LIN {X 0,Y 354.811,Z 376.286,A -85,B 0,C 180,E1 -13642.402,E2 -13642.402} C_VEL
LIN {X 0,Y 354.817,Z 376.286,A -85,B 0,C 180,E1 -13644.524,E2 -13644.524} C_VEL
LIN {X 0,Y 354.143,Z 376.373,A -85,B 0,C 180,E1 -13645.473,E2 -13645.473} C_VEL
LIN {X 0,Y 351.322,Z 376.725,A -85,B 0,C 180,E1 -13647.018,E2 -13647.018} C_VEL
LIN {X 0,Y 348.61,Z 377.585,A -85,B 0,C 180,E1 -13648.572,E2 -13648.572} C_VEL
LIN {X 0,Y 348.11,Z 378.744,A -85,B 0,C 180,E1 -13649.518,E2 -13649.518} C_VEL
LIN {X 0,Y 347.833,Z 384.152,A -85,B 0,C 180,E1 -13652.752,E2 -13652.752} C_VEL
LIN {X 0,Y 347.434,Z 390.956,A -85,B 0,C 180,E1 -13656.768,E2 -13656.768} C_VEL
LIN {X 0,Y 347.187,Z 397.381,A -85,B 0,C 180,E1 -13660.488,E2 -13660.488} C_VEL
LIN {X 0,Y 346.96,Z 403.814,A -85,B 0,C 180,E1 -13664.13,E2 -13664.13} C_VEL
LIN {X 0,Y 346.774,Z 410.819,A -85,B 0,C 180,E1 -13668.01,E2 -13668.01} C_VEL
LIN {X 0,Y 346.782,Z 411.483,A -85,B 0,C 180,E1 -13668.27,E2 -13668.27} C_VEL
LIN {X 0,Y 348.09,Z 422.89,A -85,B 0,C 180,E1 -13669.015,E2 -13669.015} C_VEL
LIN {X 0,Y 348.747,Z 429.335,A -85,B 0,C 180,E1 -13669.55,E2 -13669.55} C_VEL
LIN {X 0,Y 348.245,Z 439.424,A -85,B 0,C 180,E1 -13670.562,E2 -13670.562} C_VEL
LIN {X 0,Y 347.847,Z 448.426,A -85,B 0,C 180,E1 -13671.723,E2 -13671.723} C_VEL
LIN {X 0,Y 347.615,Z 456.417,A -85,B 0,C 180,E1 -13673.032,E2 -13673.032} C_VEL
LIN {X 0,Y 347.324,Z 463.366,A -85,B 0,C 180,E1 -13674.484,E2 -13674.484} C_VEL
LIN {X 0,Y 347.115,Z 468.718,A -85,B 0,C 180,E1 -13675.936,E2 -13675.936} C_VEL
LIN {X 0,Y 346.768,Z 473.44,A -85,B 0,C 180,E1 -13677.677,E2 -13677.677} C_VEL
LIN {X 0,Y 346.735,Z 475.64,A -85,B 0,C 180,E1 -13678.839,E2 -13678.839} C_VEL
LIN {X 0,Y 346.756,Z 477.156,A -85,B 0,C 180,E1 -13680,E2 -13680} C_VEL
LIN {X 0,Y 346.825,Z 478.018,A -85,B 0,C 180,E1 -13681.161,E2 -13681.161} C_VEL
LIN {X 0,Y 346.995,Z 478.228,A -85,B 0,C 180,E1 -13682.322,E2 -13682.322} C_VEL
LIN {X 0,Y 347.302,Z 477.789,A -85,B 0,C 180,E1 -13683.48,E2 -13683.48} C_VEL
LIN {X 0,Y 347.777,Z 476.691,A -85,B 0,C 180,E1 -13684.636,E2 -13684.636} C_VEL
LIN {X 0,Y 348.649,Z 473.789,A -85,B 0,C 180,E1 -13686.365,E2 -13686.365} C_VEL
LIN {X 0,Y 349.587,Z 469.338,A -85,B 0,C 180,E1 -13688.09,E2 -13688.09} C_VEL
LIN {X 0,Y 350.585,Z 464.252,A -85,B 0,C 180,E1 -13689.52,E2 -13689.52} C_VEL
LIN {X 0,Y 351.785,Z 457.649,A -85,B 0,C 180,E1 -13690.941,E2 -13690.941} C_VEL
LIN {X 0,Y 353.113,Z 449.6,A -85,B 0,C 180,E1 -13692.289,E2 -13692.289} C_VEL
LIN {X 0,Y 354.289,Z 439.873,A -85,B 0,C 180,E1 -13693.587,E2 -13693.587} C_VEL
LIN {X 0,Y 352.987,Z 431.307,A -85,B 0,C 180,E1 -13694.705,E2 -13694.705} C_VEL
LIN {X 0,Y 349.84,Z 420.355,A -85,B 0,C 180,E1 -13696.038,E2 -13696.038} C_VEL
LIN {X 0,Y 348.708,Z 416.833,A -85,B 0,C 180,E1 -13696.465,E2 -13696.465} C_VEL
LIN {X 0,Y 349.163,Z 413.41,A -85,B 0,C 180,E1 -13698.91,E2 -13698.91} C_VEL
LIN {X 0,Y 349.782,Z 408.791,A -85,B 0,C 180,E1 -13702.443,E2 -13702.443} C_VEL
LIN {X 0,Y 350.665,Z 404.335,A -85,B 0,C 180,E1 -13706.163,E2 -13706.163} C_VEL
LIN {X 0,Y 351.349,Z 401.637,A -85,B 0,C 180,E1 -13708.69,E2 -13708.69} C_VEL
LIN {X 0,Y 351.882,Z 399.265,A -85,B 0,C 180,E1 -13711.285,E2 -13711.285} C_VEL
LIN {X 0,Y 352.025,Z 397.313,A -85,B 0,C 180,E1 -13713.987,E2 -13713.987} C_VEL
LIN {X 0,Y 352.035,Z 395.851,A -85,B 0,C 180,E1 -13717.007,E2 -13717.007} C_VEL
LIN {X 0,Y 352.049,Z 395.224,A -85,B 0,C 180,E1 -13719.704,E2 -13719.704} C_VEL
LIN {X 0,Y 352.23,Z 395.281,A -85,B 0,C 180,E1 -13722.719,E2 -13722.719} C_VEL
LIN {X 0,Y 352.561,Z 396.33,A -85,B 0,C 180,E1 -13725.859,E2 -13725.859} C_VEL
LIN {X 0,Y 353.162,Z 398.551,A -85,B 0,C 180,E1 -13729.131,E2 -13729.131} C_VEL
LIN {X 0,Y 353.976,Z 402.286,A -85,B 0,C 180,E1 -13732.578,E2 -13732.578} C_VEL
LIN {X 0,Y 355.113,Z 406.755,A -85,B 0,C 180,E1 -13735.665,E2 -13735.665} C_VEL
LIN {X 0,Y 355.806,Z 411.281,A -85,B 0,C 180,E1 -13738.141,E2 -13738.141} C_VEL
LIN {X 0,Y 355.791,Z 413.274,A -85,B 0,C 180,E1 -13739.097,E2 -13739.097} C_VEL
LIN {X 0,Y 354.038,Z 419.488,A -85,B 0,C 180,E1 -13741.548,E2 -13741.548} C_VEL
LIN {X 0,Y 351.605,Z 429.59,A -85,B 0,C 180,E1 -13745.181,E2 -13745.181} C_VEL
LIN {X 0,Y 350.041,Z 439.051,A -85,B 0,C 180,E1 -13748.273,E2 -13748.273} C_VEL
LIN {X 0,Y 352.668,Z 451.93,A -85,B 0,C 180,E1 -13749.147,E2 -13749.147} C_VEL
LIN {X 0,Y 353.713,Z 462.761,A -85,B 0,C 180,E1 -13749.95,E2 -13749.95} C_VEL
LIN {X 0,Y 353.653,Z 473.701,A -85,B 0,C 180,E1 -13750.859,E2 -13750.859} C_VEL
LIN {X 0,Y 352.881,Z 482.708,A -85,B 0,C 180,E1 -13751.719,E2 -13751.719} C_VEL
LIN {X 0,Y 351.276,Z 493.812,A -85,B 0,C 180,E1 -13752.986,E2 -13752.986} C_VEL
LIN {X 0,Y 350.022,Z 502.896,A -85,B 0,C 180,E1 -13754.272,E2 -13754.272} C_VEL
LIN {X 0,Y 348.637,Z 512.75,A -85,B 0,C 180,E1 -13756.001,E2 -13756.001} C_VEL
LIN {X 0,Y 347.733,Z 520.726,A -85,B 0,C 180,E1 -13757.748,E2 -13757.748} C_VEL
LIN {X 0,Y 346.937,Z 527.128,A -85,B 0,C 180,E1 -13759.495,E2 -13759.495} C_VEL
LIN {X 0,Y 346.618,Z 532.253,A -85,B 0,C 180,E1 -13761.253,E2 -13761.253} C_VEL
LIN {X 0,Y 346.518,Z 536.239,A -85,B 0,C 180,E1 -13763.01,E2 -13763.01} C_VEL
LIN {X 0,Y 346.434,Z 538.314,A -85,B 0,C 180,E1 -13764.178,E2 -13764.178} C_VEL
LIN {X 0,Y 346.456,Z 539.912,A -85,B 0,C 180,E1 -13765.346,E2 -13765.346} C_VEL
LIN {X 0,Y 346.562,Z 541.078,A -85,B 0,C 180,E1 -13766.512,E2 -13766.512} C_VEL
LIN {X 0,Y 346.686,Z 541.834,A -85,B 0,C 180,E1 -13767.676,E2 -13767.676} C_VEL
LIN {X 0,Y 346.736,Z 542.119,A -85,B 0,C 180,E1 -13768.838,E2 -13768.838} C_VEL
LIN {X 0,Y 346.701,Z 541.952,A -85,B 0,C 180,E1 -13770,E2 -13770} C_VEL
LIN {X 0,Y 346.742,Z 541.378,A -85,B 0,C 180,E1 -13771.161,E2 -13771.161} C_VEL
LIN {X 0,Y 346.843,Z 540.334,A -85,B 0,C 180,E1 -13772.322,E2 -13772.322} C_VEL
LIN {X 0,Y 346.663,Z 537.849,A -85,B 0,C 180,E1 -13774.069,E2 -13774.069} C_VEL
LIN {X 0,Y 346.68,Z 534.253,A -85,B 0,C 180,E1 -13775.817,E2 -13775.817} C_VEL
LIN {X 0,Y 346.696,Z 529.411,A -85,B 0,C 180,E1 -13777.571,E2 -13777.571} C_VEL
LIN {X 0,Y 346.803,Z 523.174,A -85,B 0,C 180,E1 -13779.33,E2 -13779.33} C_VEL
LIN {X 0,Y 347.185,Z 515.215,A -85,B 0,C 180,E1 -13781.087,E2 -13781.087} C_VEL
LIN {X 0,Y 347.646,Z 507.003,A -85,B 0,C 180,E1 -13782.552,E2 -13782.552} C_VEL
LIN {X 0,Y 348.191,Z 497.967,A -85,B 0,C 180,E1 -13783.868,E2 -13783.868} C_VEL
LIN {X 0,Y 349.095,Z 486.732,A -85,B 0,C 180,E1 -13785.172,E2 -13785.172} C_VEL
LIN {X 0,Y 349.774,Z 475.649,A -85,B 0,C 180,E1 -13786.188,E2 -13786.188} C_VEL
LIN {X 0,Y 349.71,Z 468.549,A -85,B 0,C 180,E1 -13786.716,E2 -13786.716} C_VEL
LIN {X 0,Y 348.833,Z 456.7,A -85,B 0,C 180,E1 -13787.439,E2 -13787.439} C_VEL
LIN {X 0,Y 347.966,Z 443.814,A -85,B 0,C 180,E1 -13787.984,E2 -13787.984} C_VEL
LIN {X 0,Y 347.834,Z 441.173,A -85,B 0,C 180,E1 -13788.069,E2 -13788.069} C_VEL
LIN {X 0,Y 349.271,Z 426.512,A -85,B 0,C 180,E1 -13792.477,E2 -13792.477} C_VEL
LIN {X 0,Y 350.954,Z 413.38,A -85,B 0,C 180,E1 -13796.459,E2 -13796.459} C_VEL
LIN {X 0,Y 352.597,Z 402.157,A -85,B 0,C 180,E1 -13799.888,E2 -13799.888} C_VEL
LIN {X 0,Y 352.293,Z 398.982,A -85,B 0,C 180,E1 -13800.927,E2 -13800.927} C_VEL
LIN {X 0,Y 350.071,Z 388.247,A -85,B 0,C 180,E1 -13804.602,E2 -13804.602} C_VEL
LIN {X 0,Y 347.956,Z 377.826,A -85,B 0,C 180,E1 -13808.342,E2 -13808.342} C_VEL
LIN {X 0,Y 347.798,Z 377.161,A -85,B 0,C 180,E1 -13808.68,E2 -13808.68} C_VEL
LIN {X 0,Y 347.752,Z 377.169,A -85,B 0,C 180,E1 -13811.83,E2 -13811.83} C_VEL
LIN {X 0,Y 347.767,Z 377.164,A -85,B 0,C 180,E1 -13815.017,E2 -13815.017} C_VEL
LIN {X 0,Y 347.758,Z 377.168,A -85,B 0,C 180,E1 -13818.396,E2 -13818.396} C_VEL
LIN {X 0,Y 347.775,Z 377.167,A -85,B 0,C 180,E1 -13822.011,E2 -13822.011} C_VEL
LIN {X 0,Y 347.745,Z 377.167,A -85,B 0,C 180,E1 -13825.536,E2 -13825.536} C_VEL
LIN {X 0,Y 347.746,Z 377.169,A -85,B 0,C 180,E1 -13828.3,E2 -13828.3} C_VEL
LIN {X 0,Y 347.779,Z 377.161,A -85,B 0,C 180,E1 -13830.988,E2 -13830.988} C_VEL
LIN {X 0,Y 347.832,Z 377.158,A -85,B 0,C 180,E1 -13833.608,E2 -13833.608} C_VEL
LIN {X 0,Y 347.789,Z 377.164,A -85,B 0,C 180,E1 -13836.162,E2 -13836.162} C_VEL
LIN {X 0,Y 347.818,Z 377.162,A -85,B 0,C 180,E1 -13839.91,E2 -13839.91} C_VEL
LIN {X 0,Y 347.867,Z 377.151,A -85,B 0,C 180,E1 -13842.359,E2 -13842.359} C_VEL
LIN {X 0,Y 347.898,Z 377.151,A -85,B 0,C 180,E1 -13845.971,E2 -13845.971} C_VEL
LIN {X 0,Y 347.929,Z 377.147,A -85,B 0,C 180,E1 -13849.526,E2 -13849.526} C_VEL
LIN {X 0,Y 348.075,Z 377.128,A -85,B 0,C 180,E1 -13851.875,E2 -13851.875} C_VEL
LIN {X 0,Y 348.069,Z 377.126,A -85,B 0,C 180,E1 -13854.206,E2 -13854.206} C_VEL
LIN {X 0,Y 348.209,Z 377.113,A -85,B 0,C 180,E1 -13857.687,E2 -13857.687} C_VEL
LIN {X 0,Y 348.347,Z 377.092,A -85,B 0,C 180,E1 -13860,E2 -13860} C_VEL
LIN {X 0,Y 348.207,Z 377.108,A -85,B 0,C 180,E1 -13862.314,E2 -13862.314} C_VEL
LIN {X 0,Y 348.108,Z 377.123,A -85,B 0,C 180,E1 -13866.958,E2 -13866.958} C_VEL
LIN {X 0,Y 347.97,Z 377.143,A -85,B 0,C 180,E1 -13869.299,E2 -13869.299} C_VEL
LIN {X 0,Y 347.895,Z 377.149,A -85,B 0,C 180,E1 -13872.839,E2 -13872.839} C_VEL
LIN {X 0,Y 347.84,Z 377.154,A -85,B 0,C 180,E1 -13876.431,E2 -13876.431} C_VEL
LIN {X 0,Y 347.852,Z 377.155,A -85,B 0,C 180,E1 -13878.861,E2 -13878.861} C_VEL
LIN {X 0,Y 347.775,Z 377.163,A -85,B 0,C 180,E1 -13882.579,E2 -13882.579} C_VEL
LIN {X 0,Y 347.814,Z 377.163,A -85,B 0,C 180,E1 -13885.108,E2 -13885.108} C_VEL
LIN {X 0,Y 347.81,Z 377.158,A -85,B 0,C 180,E1 -13887.694,E2 -13887.694} C_VEL
LIN {X 0,Y 347.764,Z 377.164,A -85,B 0,C 180,E1 -13890.347,E2 -13890.347} C_VEL
LIN {X 0,Y 347.745,Z 377.168,A -85,B 0,C 180,E1 -13894.464,E2 -13894.464} C_VEL
LIN {X 0,Y 347.775,Z 377.162,A -85,B 0,C 180,E1 -13897.989,E2 -13897.989} C_VEL
LIN {X 0,Y 347.751,Z 377.165,A -85,B 0,C 180,E1 -13901.83,E2 -13901.83} C_VEL
LIN {X 0,Y 347.766,Z 377.166,A -85,B 0,C 180,E1 -13905.017,E2 -13905.017} C_VEL
LIN {X 0,Y 347.752,Z 377.168,A -85,B 0,C 180,E1 -13908.397,E2 -13908.397} C_VEL
LIN {X 0,Y 347.777,Z 377.163,A -85,B 0,C 180,E1 -13912.011,E2 -13912.011} C_VEL
LIN {X 0,Y 347.745,Z 377.166,A -85,B 0,C 180,E1 -13915.536,E2 -13915.536} C_VEL
LIN {X 0,Y 347.746,Z 377.169,A -85,B 0,C 180,E1 -13918.301,E2 -13918.301} C_VEL
LIN {X 0,Y 347.78,Z 377.163,A -85,B 0,C 180,E1 -13920.988,E2 -13920.988} C_VEL
LIN {X 0,Y 347.832,Z 377.155,A -85,B 0,C 180,E1 -13923.608,E2 -13923.608} C_VEL
LIN {X 0,Y 347.791,Z 377.164,A -85,B 0,C 180,E1 -13926.162,E2 -13926.162} C_VEL
LIN {X 0,Y 347.83,Z 377.157,A -85,B 0,C 180,E1 -13929.911,E2 -13929.911} C_VEL
LIN {X 0,Y 347.87,Z 377.155,A -85,B 0,C 180,E1 -13932.36,E2 -13932.36} C_VEL
LIN {X 0,Y 347.899,Z 377.15,A -85,B 0,C 180,E1 -13935.971,E2 -13935.971} C_VEL
LIN {X 0,Y 347.932,Z 377.143,A -85,B 0,C 180,E1 -13939.526,E2 -13939.526} C_VEL
LIN {X 0,Y 348.094,Z 377.122,A -85,B 0,C 180,E1 -13943.042,E2 -13943.042} C_VEL
LIN {X 0,Y 348.209,Z 377.111,A -85,B 0,C 180,E1 -13947.687,E2 -13947.687} C_VEL
LIN {X 0,Y 348.37,Z 377.093,A -85,B 0,C 180,E1 -13950,E2 -13950} C_VEL
LIN {X 0,Y 348.209,Z 377.11,A -85,B 0,C 180,E1 -13952.314,E2 -13952.314} C_VEL
LIN {X 0,Y 348.093,Z 377.122,A -85,B 0,C 180,E1 -13956.958,E2 -13956.958} C_VEL
LIN {X 0,Y 347.932,Z 377.143,A -85,B 0,C 180,E1 -13960.475,E2 -13960.475} C_VEL
LIN {X 0,Y 347.901,Z 377.148,A -85,B 0,C 180,E1 -13964.15,E2 -13964.15} C_VEL
LIN {X 0,Y 347.894,Z 377.148,A -85,B 0,C 180,E1 -13968.291,E2 -13968.291} C_VEL
LIN {X 0,Y 347.792,Z 377.165,A -85,B 0,C 180,E1 -13971.635,E2 -13971.635} C_VEL
LIN {X 0,Y 347.815,Z 377.158,A -85,B 0,C 180,E1 -13975.109,E2 -13975.109} C_VEL
LIN {X 0,Y 347.811,Z 377.162,A -85,B 0,C 180,E1 -13977.694,E2 -13977.694} C_VEL
LIN {X 0,Y 347.752,Z 377.165,A -85,B 0,C 180,E1 -13980.348,E2 -13980.348} C_VEL
LIN {X 0,Y 347.751,Z 377.166,A -85,B 0,C 180,E1 -13984.044,E2 -13984.044} C_VEL
LIN {X 0,Y 347.768,Z 377.168,A -85,B 0,C 180,E1 -13987.32,E2 -13987.32} C_VEL
LIN {X 0,Y 347.735,Z 377.167,A -85,B 0,C 180,E1 -13990.297,E2 -13990.297} C_VEL
LIN {X 0,Y 347.726,Z 377.173,A -85,B 0,C 180,E1 -13993.408,E2 -13993.408} C_VEL
LIN {X 0,Y 347.73,Z 377.169,A -85,B 0,C 180,E1 -13996.686,E2 -13996.686} C_VEL
LIN {X 0,Y 347.75,Z 377.165,A -85,B 0,C 180,E1 -14000.173,E2 -14000.173} C_VEL
LIN {X 0,Y 347.765,Z 377.165,A -85,B 0,C 180,E1 -14002.679,E2 -14002.679} C_VEL
LIN {X 0,Y 347.766,Z 377.163,A -85,B 0,C 180,E1 -14005.953,E2 -14005.953} C_VEL
LIN {X 0,Y 347.954,Z 377.227,A -85,B 0,C 180,E1 -14008.576,E2 -14008.576} C_VEL
LIN {X 0,Y 348.11,Z 378.744,A -85,B 0,C 180,E1 -14009.518,E2 -14009.518} C_VEL
LIN {X 0,Y 347.558,Z 380.345,A -85,B 0,C 180,E1 -14010.446,E2 -14010.446} C_VEL
LIN {X 0,Y 345.96,Z 382.043,A -85,B 0,C 180,E1 -14011.349,E2 -14011.349} C_VEL
LIN {X 0,Y 341.976,Z 385.511,A -85,B 0,C 180,E1 -14013.146,E2 -14013.146} C_VEL
LIN {X 0,Y 340.757,Z 387.216,A -85,B 0,C 180,E1 -14014.086,E2 -14014.086} C_VEL
LIN {X 0,Y 340.618,Z 387.767,A -85,B 0,C 180,E1 -14014.408,E2 -14014.408} C_VEL
LIN {X 0,Y 340.259,Z 394.446,A -85,B 0,C 180,E1 -14018.353,E2 -14018.353} C_VEL
LIN {X 0,Y 340.044,Z 400.608,A -85,B 0,C 180,E1 -14021.94,E2 -14021.94} C_VEL
LIN {X 0,Y 339.801,Z 407.099,A -85,B 0,C 180,E1 -14025.629,E2 -14025.629} C_VEL
LIN {X 0,Y 339.711,Z 411.711,A -85,B 0,C 180,E1 -14028.136,E2 -14028.136} C_VEL
LIN {X 0,Y 340.876,Z 422.632,A -85,B 0,C 180,E1 -14028.855,E2 -14028.855} C_VEL
LIN {X 0,Y 341.674,Z 430.029,A -85,B 0,C 180,E1 -14029.481,E2 -14029.481} C_VEL
LIN {X 0,Y 341.165,Z 440.077,A -85,B 0,C 180,E1 -14030.514,E2 -14030.514} C_VEL
LIN {X 0,Y 340.766,Z 449.071,A -85,B 0,C 180,E1 -14031.699,E2 -14031.699} C_VEL
LIN {X 0,Y 340.484,Z 457.854,A -85,B 0,C 180,E1 -14033.184,E2 -14033.184} C_VEL
LIN {X 0,Y 340.215,Z 464.634,A -85,B 0,C 180,E1 -14034.666,E2 -14034.666} C_VEL
LIN {X 0,Y 340.056,Z 468.902,A -85,B 0,C 180,E1 -14035.852,E2 -14035.852} C_VEL
LIN {X 0,Y 339.706,Z 473.771,A -85,B 0,C 180,E1 -14037.629,E2 -14037.629} C_VEL
LIN {X 0,Y 339.66,Z 476.091,A -85,B 0,C 180,E1 -14038.814,E2 -14038.814} C_VEL
LIN {X 0,Y 339.708,Z 477.725,A -85,B 0,C 180,E1 -14040,E2 -14040} C_VEL
LIN {X 0,Y 339.779,Z 478.706,A -85,B 0,C 180,E1 -14041.185,E2 -14041.185} C_VEL
LIN {X 0,Y 339.956,Z 479.035,A -85,B 0,C 180,E1 -14042.37,E2 -14042.37} C_VEL
LIN {X 0,Y 340.276,Z 478.708,A -85,B 0,C 180,E1 -14043.552,E2 -14043.552} C_VEL
LIN {X 0,Y 340.777,Z 477.733,A -85,B 0,C 180,E1 -14044.732,E2 -14044.732} C_VEL
LIN {X 0,Y 341.718,Z 475.035,A -85,B 0,C 180,E1 -14046.495,E2 -14046.495} C_VEL
LIN {X 0,Y 342.707,Z 470.797,A -85,B 0,C 180,E1 -14048.253,E2 -14048.253} C_VEL
LIN {X 0,Y 343.762,Z 465.894,A -85,B 0,C 180,E1 -14049.71,E2 -14049.71} C_VEL
LIN {X 0,Y 345.018,Z 459.627,A -85,B 0,C 180,E1 -14051.158,E2 -14051.158} C_VEL
LIN {X 0,Y 346.492,Z 451.602,A -85,B 0,C 180,E1 -14052.594,E2 -14052.594} C_VEL
LIN {X 0,Y 347.833,Z 442.717,A -85,B 0,C 180,E1 -14053.844,E2 -14053.844} C_VEL
LIN {X 0,Y 347.019,Z 435.357,A -85,B 0,C 180,E1 -14054.868,E2 -14054.868} C_VEL
LIN {X 0,Y 344.892,Z 426.575,A -85,B 0,C 180,E1 -14056.044,E2 -14056.044} C_VEL
LIN {X 0,Y 341.879,Z 417.464,A -85,B 0,C 180,E1 -14057.188,E2 -14057.188} C_VEL
LIN {X 0,Y 342.49,Z 413.167,A -85,B 0,C 180,E1 -14060.417,E2 -14060.417} C_VEL
LIN {X 0,Y 343.282,Z 408.574,A -85,B 0,C 180,E1 -14064.171,E2 -14064.171} C_VEL
LIN {X 0,Y 343.97,Z 405.739,A -85,B 0,C 180,E1 -14066.712,E2 -14066.712} C_VEL
LIN {X 0,Y 344.7,Z 403.141,A -85,B 0,C 180,E1 -14069.297,E2 -14069.297} C_VEL
LIN {X 0,Y 345.101,Z 401.496,A -85,B 0,C 180,E1 -14071.203,E2 -14071.203} C_VEL
LIN {X 0,Y 345.285,Z 399.912,A -85,B 0,C 180,E1 -14073.433,E2 -14073.433} C_VEL
LIN {X 0,Y 345.312,Z 398.566,A -85,B 0,C 180,E1 -14076.173,E2 -14076.173} C_VEL
LIN {X 0,Y 345.376,Z 397.718,A -85,B 0,C 180,E1 -14079.352,E2 -14079.352} C_VEL
LIN {X 0,Y 345.53,Z 397.719,A -85,B 0,C 180,E1 -14082.161,E2 -14082.161} C_VEL
LIN {X 0,Y 345.855,Z 398.65,A -85,B 0,C 180,E1 -14085.335,E2 -14085.335} C_VEL
LIN {X 0,Y 346.43,Z 400.728,A -85,B 0,C 180,E1 -14088.644,E2 -14088.644} C_VEL
LIN {X 0,Y 347.202,Z 404.263,A -85,B 0,C 180,E1 -14092.133,E2 -14092.133} C_VEL
LIN {X 0,Y 348.153,Z 407.982,A -85,B 0,C 180,E1 -14094.878,E2 -14094.878} C_VEL
LIN {X 0,Y 348.995,Z 412.834,A -85,B 0,C 180,E1 -14097.757,E2 -14097.757} C_VEL
LIN {X 0,Y 348.938,Z 415.579,A -85,B 0,C 180,E1 -14099.096,E2 -14099.096} C_VEL
LIN {X 0,Y 346.621,Z 423.381,A -85,B 0,C 180,E1 -14102.203,E2 -14102.203} C_VEL
LIN {X 0,Y 344.246,Z 433.589,A -85,B 0,C 180,E1 -14105.901,E2 -14105.901} C_VEL
LIN {X 0,Y 343.379,Z 438.444,A -85,B 0,C 180,E1 -14107.552,E2 -14107.552} C_VEL
LIN {X 0,Y 346.233,Z 452.39,A -85,B 0,C 180,E1 -14108.569,E2 -14108.569} C_VEL
LIN {X 0,Y 347.303,Z 464.156,A -85,B 0,C 180,E1 -14109.51,E2 -14109.51} C_VEL
LIN {X 0,Y 347.102,Z 475.082,A -85,B 0,C 180,E1 -14110.483,E2 -14110.483} C_VEL
LIN {X 0,Y 345.846,Z 486.319,A -85,B 0,C 180,E1 -14111.64,E2 -14111.64} C_VEL
LIN {X 0,Y 344.26,Z 496.517,A -85,B 0,C 180,E1 -14112.934,E2 -14112.934} C_VEL
LIN {X 0,Y 342.655,Z 506.7,A -85,B 0,C 180,E1 -14114.536,E2 -14114.536} C_VEL
LIN {X 0,Y 341.399,Z 515.616,A -85,B 0,C 180,E1 -14116.306,E2 -14116.306} C_VEL
LIN {X 0,Y 340.431,Z 522.882,A -85,B 0,C 180,E1 -14118.086,E2 -14118.086} C_VEL
LIN {X 0,Y 339.772,Z 528.693,A -85,B 0,C 180,E1 -14119.873,E2 -14119.873} C_VEL
LIN {X 0,Y 339.466,Z 533.309,A -85,B 0,C 180,E1 -14121.667,E2 -14121.667} C_VEL
LIN {X 0,Y 339.394,Z 537.225,A -85,B 0,C 180,E1 -14123.701,E2 -14123.701} C_VEL
LIN {X 0,Y 339.383,Z 539.319,A -85,B 0,C 180,E1 -14125.248,E2 -14125.248} C_VEL
LIN {X 0,Y 339.469,Z 540.442,A -85,B 0,C 180,E1 -14126.439,E2 -14126.439} C_VEL
LIN {X 0,Y 339.614,Z 541.139,A -85,B 0,C 180,E1 -14127.628,E2 -14127.628} C_VEL
LIN {X 0,Y 339.69,Z 541.36,A -85,B 0,C 180,E1 -14128.814,E2 -14128.814} C_VEL
LIN {X 0,Y 339.656,Z 541.154,A -85,B 0,C 180,E1 -14130,E2 -14130} C_VEL
LIN {X 0,Y 339.7,Z 540.518,A -85,B 0,C 180,E1 -14131.185,E2 -14131.185} C_VEL
LIN {X 0,Y 339.797,Z 539.4,A -85,B 0,C 180,E1 -14132.371,E2 -14132.371} C_VEL
LIN {X 0,Y 339.612,Z 536.816,A -85,B 0,C 180,E1 -14134.153,E2 -14134.153} C_VEL
LIN {X 0,Y 339.624,Z 533.114,A -85,B 0,C 180,E1 -14135.939,E2 -14135.939} C_VEL
LIN {X 0,Y 339.635,Z 528.154,A -85,B 0,C 180,E1 -14137.73,E2 -14137.73} C_VEL
LIN {X 0,Y 339.77,Z 521.722,A -85,B 0,C 180,E1 -14139.525,E2 -14139.525} C_VEL
LIN {X 0,Y 340.163,Z 513.592,A -85,B 0,C 180,E1 -14141.319,E2 -14141.319} C_VEL
LIN {X 0,Y 340.696,Z 505.172,A -85,B 0,C 180,E1 -14142.812,E2 -14142.812} C_VEL
LIN {X 0,Y 341.276,Z 495.815,A -85,B 0,C 180,E1 -14144.155,E2 -14144.155} C_VEL
LIN {X 0,Y 342.11,Z 485.373,A -85,B 0,C 180,E1 -14145.368,E2 -14145.368} C_VEL
LIN {X 0,Y 342.744,Z 474.39,A -85,B 0,C 180,E1 -14146.376,E2 -14146.376} C_VEL
LIN {X 0,Y 342.379,Z 464.766,A -85,B 0,C 180,E1 -14147.085,E2 -14147.085} C_VEL
LIN {X 0,Y 341.335,Z 450.937,A -85,B 0,C 180,E1 -14147.854,E2 -14147.854} C_VEL
LIN {X 0,Y 340.8,Z 440.896,A -85,B 0,C 180,E1 -14148.245,E2 -14148.245} C_VEL
LIN {X 0,Y 342.397,Z 425.635,A -85,B 0,C 180,E1 -14152.954,E2 -14152.954} C_VEL
LIN {X 0,Y 344.274,Z 411.567,A -85,B 0,C 180,E1 -14157.343,E2 -14157.343} C_VEL
LIN {X 0,Y 345.567,Z 403.489,A -85,B 0,C 180,E1 -14159.885,E2 -14159.885} C_VEL
LIN {X 0,Y 345.543,Z 401.404,A -85,B 0,C 180,E1 -14160.562,E2 -14160.562} C_VEL
LIN {X 0,Y 343.363,Z 390.864,A -85,B 0,C 180,E1 -14164.22,E2 -14164.22} C_VEL
LIN {X 0,Y 341.152,Z 380.028,A -85,B 0,C 180,E1 -14168.172,E2 -14168.172} C_VEL
LIN {X 0,Y 340.739,Z 378.04,A -85,B 0,C 180,E1 -14168.951,E2 -14168.951} C_VEL
LIN {X 0,Y 340.69,Z 378.045,A -85,B 0,C 180,E1 -14172.902,E2 -14172.902} C_VEL
LIN {X 0,Y 340.667,Z 378.052,A -85,B 0,C 180,E1 -14176.224,E2 -14176.224} C_VEL
LIN {X 0,Y 340.7,Z 378.045,A -85,B 0,C 180,E1 -14179.751,E2 -14179.751} C_VEL
LIN {X 0,Y 340.706,Z 378.043,A -85,B 0,C 180,E1 -14183.258,E2 -14183.258} C_VEL
LIN {X 0,Y 340.695,Z 378.049,A -85,B 0,C 180,E1 -14186.154,E2 -14186.154} C_VEL
LIN {X 0,Y 340.742,Z 378.04,A -85,B 0,C 180,E1 -14190.329,E2 -14190.329} C_VEL
LIN {X 0,Y 340.804,Z 378.03,A -85,B 0,C 180,E1 -14193.02,E2 -14193.02} C_VEL
LIN {X 0,Y 340.757,Z 378.039,A -85,B 0,C 180,E1 -14195.638,E2 -14195.638} C_VEL
LIN {X 0,Y 340.749,Z 378.04,A -85,B 0,C 180,E1 -14199.474,E2 -14199.474} C_VEL
LIN {X 0,Y 340.859,Z 378.027,A -85,B 0,C 180,E1 -14201.984,E2 -14201.984} C_VEL
LIN {X 0,Y 340.87,Z 378.027,A -85,B 0,C 180,E1 -14205.705,E2 -14205.705} C_VEL
LIN {X 0,Y 340.872,Z 378.024,A -85,B 0,C 180,E1 -14209.306,E2 -14209.306} C_VEL
LIN {X 0,Y 341.077,Z 377.996,A -85,B 0,C 180,E1 -14212.898,E2 -14212.898} C_VEL
LIN {X 0,Y 341.171,Z 377.989,A -85,B 0,C 180,E1 -14217.639,E2 -14217.639} C_VEL
LIN {X 0,Y 341.298,Z 377.97,A -85,B 0,C 180,E1 -14220,E2 -14220} C_VEL
LIN {X 0,Y 341.169,Z 377.985,A -85,B 0,C 180,E1 -14222.361,E2 -14222.361} C_VEL
LIN {X 0,Y 341.077,Z 377.999,A -85,B 0,C 180,E1 -14227.102,E2 -14227.102} C_VEL
LIN {X 0,Y 340.876,Z 378.022,A -85,B 0,C 180,E1 -14230.694,E2 -14230.694} C_VEL
LIN {X 0,Y 340.863,Z 378.023,A -85,B 0,C 180,E1 -14234.325,E2 -14234.325} C_VEL
LIN {X 0,Y 340.837,Z 378.026,A -85,B 0,C 180,E1 -14238.466,E2 -14238.466} C_VEL
LIN {X 0,Y 340.754,Z 378.037,A -85,B 0,C 180,E1 -14241.857,E2 -14241.857} C_VEL
LIN {X 0,Y 340.773,Z 378.035,A -85,B 0,C 180,E1 -14245.664,E2 -14245.664} C_VEL
LIN {X 0,Y 340.741,Z 378.038,A -85,B 0,C 180,E1 -14248.32,E2 -14248.32} C_VEL
LIN {X 0,Y 340.704,Z 378.048,A -85,B 0,C 180,E1 -14251.044,E2 -14251.044} C_VEL
LIN {X 0,Y 340.719,Z 378.043,A -85,B 0,C 180,E1 -14255.279,E2 -14255.279} C_VEL
LIN {X 0,Y 340.711,Z 378.043,A -85,B 0,C 180,E1 -14258.386,E2 -14258.386} C_VEL
LIN {X 0,Y 340.7,Z 378.044,A -85,B 0,C 180,E1 -14262.046,E2 -14262.046} C_VEL
LIN {X 0,Y 340.683,Z 378.046,A -85,B 0,C 180,E1 -14265.461,E2 -14265.461} C_VEL
LIN {X 0,Y 340.688,Z 378.05,A -85,B 0,C 180,E1 -14268.691,E2 -14268.691} C_VEL
LIN {X 0,Y 340.736,Z 378.039,A -85,B 0,C 180,E1 -14271.773,E2 -14271.773} C_VEL
LIN {X 0,Y 340.724,Z 378.04,A -85,B 0,C 180,E1 -14275.596,E2 -14275.596} C_VEL
LIN {X 0,Y 340.699,Z 378.045,A -85,B 0,C 180,E1 -14278.956,E2 -14278.956} C_VEL
LIN {X 0,Y 340.805,Z 378.031,A -85,B 0,C 180,E1 -14283.02,E2 -14283.02} C_VEL
LIN {X 0,Y 340.732,Z 378.04,A -85,B 0,C 180,E1 -14286.928,E2 -14286.928} C_VEL
LIN {X 0,Y 340.802,Z 378.032,A -85,B 0,C 180,E1 -14290.734,E2 -14290.734} C_VEL
LIN {X 0,Y 340.791,Z 378.032,A -85,B 0,C 180,E1 -14293.219,E2 -14293.219} C_VEL
LIN {X 0,Y 340.847,Z 378.026,A -85,B 0,C 180,E1 -14296.891,E2 -14296.891} C_VEL
LIN {X 0,Y 340.929,Z 378.017,A -85,B 0,C 180,E1 -14300.508,E2 -14300.508} C_VEL
LIN {X 0,Y 341.063,Z 377.998,A -85,B 0,C 180,E1 -14302.898,E2 -14302.898} C_VEL
LIN {X 0,Y 341.171,Z 377.987,A -85,B 0,C 180,E1 -14307.639,E2 -14307.639} C_VEL
LIN {X 0,Y 341.319,Z 377.971,A -85,B 0,C 180,E1 -14310,E2 -14310} C_VEL
LIN {X 0,Y 341.171,Z 377.986,A -85,B 0,C 180,E1 -14312.361,E2 -14312.361} C_VEL
LIN {X 0,Y 341.061,Z 377.999,A -85,B 0,C 180,E1 -14317.102,E2 -14317.102} C_VEL
LIN {X 0,Y 340.874,Z 378.022,A -85,B 0,C 180,E1 -14320.694,E2 -14320.694} C_VEL
LIN {X 0,Y 340.866,Z 378.023,A -85,B 0,C 180,E1 -14324.325,E2 -14324.325} C_VEL
LIN {X 0,Y 340.841,Z 378.026,A -85,B 0,C 180,E1 -14328.467,E2 -14328.467} C_VEL
LIN {X 0,Y 340.756,Z 378.04,A -85,B 0,C 180,E1 -14331.857,E2 -14331.857} C_VEL
LIN {X 0,Y 340.775,Z 378.039,A -85,B 0,C 180,E1 -14335.664,E2 -14335.664} C_VEL
LIN {X 0,Y 340.731,Z 378.04,A -85,B 0,C 180,E1 -14338.321,E2 -14338.321} C_VEL
LIN {X 0,Y 340.7,Z 378.045,A -85,B 0,C 180,E1 -14341.045,E2 -14341.045} C_VEL
LIN {X 0,Y 340.721,Z 378.045,A -85,B 0,C 180,E1 -14345.279,E2 -14345.279} C_VEL
LIN {X 0,Y 340.714,Z 378.041,A -85,B 0,C 180,E1 -14348.387,E2 -14348.387} C_VEL
LIN {X 0,Y 340.702,Z 378.043,A -85,B 0,C 180,E1 -14352.046,E2 -14352.046} C_VEL
LIN {X 0,Y 340.687,Z 378.048,A -85,B 0,C 180,E1 -14355.462,E2 -14355.462} C_VEL
LIN {X 0,Y 340.689,Z 378.046,A -85,B 0,C 180,E1 -14358.691,E2 -14358.691} C_VEL
LIN {X 0,Y 340.736,Z 378.04,A -85,B 0,C 180,E1 -14361.773,E2 -14361.773} C_VEL
LIN {X 0,Y 340.735,Z 378.04,A -85,B 0,C 180,E1 -14365.593,E2 -14365.593} C_VEL
LIN {X 0,Y 340.918,Z 378.162,A -85,B 0,C 180,E1 -14368.546,E2 -14368.546} C_VEL
LIN {X 0,Y 341.038,Z 381.092,A -85,B 0,C 180,E1 -14370.358,E2 -14370.358} C_VEL
LIN {X 0,Y 340.633,Z 387.625,A -85,B 0,C 180,E1 -14374.324,E2 -14374.324} C_VEL
LIN {X 0,Y 340.618,Z 387.767,A -85,B 0,C 180,E1 -14374.408,E2 -14374.408} C_VEL
LIN {X 0,Y 339.816,Z 389.44,A -85,B 0,C 180,E1 -14375.353,E2 -14375.353} C_VEL
LIN {X 0,Y 336.799,Z 392.336,A -85,B 0,C 180,E1 -14376.877,E2 -14376.877} C_VEL
LIN {X 0,Y 334.301,Z 394.67,A -85,B 0,C 180,E1 -14378.111,E2 -14378.111} C_VEL
LIN {X 0,Y 333.228,Z 396.391,A -85,B 0,C 180,E1 -14379.071,E2 -14379.071} C_VEL
LIN {X 0,Y 333.137,Z 396.949,A -85,B 0,C 180,E1 -14379.398,E2 -14379.398} C_VEL
LIN {X 0,Y 332.924,Z 402.773,A -85,B 0,C 180,E1 -14382.81,E2 -14382.81} C_VEL
LIN {X 0,Y 332.704,Z 409.346,A -85,B 0,C 180,E1 -14386.564,E2 -14386.564} C_VEL
LIN {X 0,Y 332.633,Z 411.933,A -85,B 0,C 180,E1 -14387.996,E2 -14387.996} C_VEL
LIN {X 0,Y 333.839,Z 423.386,A -85,B 0,C 180,E1 -14388.771,E2 -14388.771} C_VEL
LIN {X 0,Y 334.582,Z 430.717,A -85,B 0,C 180,E1 -14389.409,E2 -14389.409} C_VEL
LIN {X 0,Y 334.081,Z 440.714,A -85,B 0,C 180,E1 -14390.464,E2 -14390.464} C_VEL
LIN {X 0,Y 333.676,Z 449.999,A -85,B 0,C 180,E1 -14391.727,E2 -14391.727} C_VEL
LIN {X 0,Y 333.436,Z 457.622,A -85,B 0,C 180,E1 -14393.039,E2 -14393.039} C_VEL
LIN {X 0,Y 333.141,Z 464.588,A -85,B 0,C 180,E1 -14394.553,E2 -14394.553} C_VEL
LIN {X 0,Y 332.98,Z 469.03,A -85,B 0,C 180,E1 -14395.764,E2 -14395.764} C_VEL
LIN {X 0,Y 332.646,Z 474.098,A -85,B 0,C 180,E1 -14397.578,E2 -14397.578} C_VEL
LIN {X 0,Y 332.587,Z 476.542,A -85,B 0,C 180,E1 -14398.789,E2 -14398.789} C_VEL
LIN {X 0,Y 332.643,Z 478.294,A -85,B 0,C 180,E1 -14400,E2 -14400} C_VEL
LIN {X 0,Y 332.733,Z 479.383,A -85,B 0,C 180,E1 -14401.21,E2 -14401.21} C_VEL
LIN {X 0,Y 332.917,Z 479.822,A -85,B 0,C 180,E1 -14402.42,E2 -14402.42} C_VEL
LIN {X 0,Y 333.248,Z 479.611,A -85,B 0,C 180,E1 -14403.627,E2 -14403.627} C_VEL
LIN {X 0,Y 333.775,Z 478.755,A -85,B 0,C 180,E1 -14404.831,E2 -14404.831} C_VEL
LIN {X 0,Y 334.785,Z 476.249,A -85,B 0,C 180,E1 -14406.63,E2 -14406.63} C_VEL
LIN {X 0,Y 335.827,Z 472.249,A -85,B 0,C 180,E1 -14408.424,E2 -14408.424} C_VEL
LIN {X 0,Y 337.22,Z 466.548,A -85,B 0,C 180,E1 -14410.204,E2 -14410.204} C_VEL
LIN {X 0,Y 338.566,Z 460.254,A -85,B 0,C 180,E1 -14411.677,E2 -14411.677} C_VEL
LIN {X 0,Y 340.161,Z 452.184,A -85,B 0,C 180,E1 -14413.136,E2 -14413.136} C_VEL
LIN {X 0,Y 341.45,Z 444.238,A -85,B 0,C 180,E1 -14414.3,E2 -14414.3} C_VEL
LIN {X 0,Y 340.39,Z 435.676,A -85,B 0,C 180,E1 -14415.57,E2 -14415.57} C_VEL
LIN {X 0,Y 337.43,Z 424.731,A -85,B 0,C 180,E1 -14417.109,E2 -14417.109} C_VEL
LIN {X 0,Y 335.159,Z 418.017,A -85,B 0,C 180,E1 -14418.017,E2 -14418.017} C_VEL
LIN {X 0,Y 335.958,Z 412.885,A -85,B 0,C 180,E1 -14422.12,E2 -14422.12} C_VEL
LIN {X 0,Y 337.031,Z 408.217,A -85,B 0,C 180,E1 -14426.276,E2 -14426.276} C_VEL
LIN {X 0,Y 337.862,Z 405.426,A -85,B 0,C 180,E1 -14429.113,E2 -14429.113} C_VEL
LIN {X 0,Y 338.404,Z 403.382,A -85,B 0,C 180,E1 -14431.625,E2 -14431.625} C_VEL
LIN {X 0,Y 338.578,Z 401.879,A -85,B 0,C 180,E1 -14434.087,E2 -14434.087} C_VEL
LIN {X 0,Y 338.633,Z 400.678,A -85,B 0,C 180,E1 -14437.004,E2 -14437.004} C_VEL
LIN {X 0,Y 338.75,Z 400.136,A -85,B 0,C 180,E1 -14440.027,E2 -14440.027} C_VEL
LIN {X 0,Y 339.042,Z 400.537,A -85,B 0,C 180,E1 -14443.488,E2 -14443.488} C_VEL
LIN {X 0,Y 339.465,Z 402.087,A -85,B 0,C 180,E1 -14446.905,E2 -14446.905} C_VEL
LIN {X 0,Y 340.054,Z 404.41,A -85,B 0,C 180,E1 -14449.88,E2 -14449.88} C_VEL
LIN {X 0,Y 340.985,Z 408.52,A -85,B 0,C 180,E1 -14453.497,E2 -14453.497} C_VEL
LIN {X 0,Y 341.925,Z 412.603,A -85,B 0,C 180,E1 -14456.291,E2 -14456.291} C_VEL
LIN {X 0,Y 342.272,Z 416.487,A -85,B 0,C 180,E1 -14458.426,E2 -14458.426} C_VEL
LIN {X 0,Y 341.52,Z 419.565,A -85,B 0,C 180,E1 -14459.803,E2 -14459.803} C_VEL
LIN {X 0,Y 338.71,Z 429.162,A -85,B 0,C 180,E1 -14463.58,E2 -14463.58} C_VEL
LIN {X 0,Y 336.82,Z 438.106,A -85,B 0,C 180,E1 -14466.791,E2 -14466.791} C_VEL
LIN {X 0,Y 339.774,Z 452.306,A -85,B 0,C 180,E1 -14467.908,E2 -14467.908} C_VEL
LIN {X 0,Y 340.881,Z 463.727,A -85,B 0,C 180,E1 -14468.884,E2 -14468.884} C_VEL
LIN {X 0,Y 340.668,Z 475.07,A -85,B 0,C 180,E1 -14469.942,E2 -14469.942} C_VEL
LIN {X 0,Y 339.565,Z 484.807,A -85,B 0,C 180,E1 -14470.975,E2 -14470.975} C_VEL
LIN {X 0,Y 337.804,Z 495.115,A -85,B 0,C 180,E1 -14472.285,E2 -14472.285} C_VEL
LIN {X 0,Y 336.111,Z 505.372,A -85,B 0,C 180,E1 -14473.915,E2 -14473.915} C_VEL
LIN {X 0,Y 334.635,Z 514.359,A -85,B 0,C 180,E1 -14475.713,E2 -14475.713} C_VEL
LIN {X 0,Y 333.651,Z 521.689,A -85,B 0,C 180,E1 -14477.531,E2 -14477.531} C_VEL
LIN {X 0,Y 332.879,Z 526.675,A -85,B 0,C 180,E1 -14479.046,E2 -14479.046} C_VEL
LIN {X 0,Y 332.501,Z 531.569,A -85,B 0,C 180,E1 -14480.878,E2 -14480.878} C_VEL
LIN {X 0,Y 332.349,Z 535.338,A -85,B 0,C 180,E1 -14482.71,E2 -14482.71} C_VEL
LIN {X 0,Y 332.289,Z 537.248,A -85,B 0,C 180,E1 -14483.929,E2 -14483.929} C_VEL
LIN {X 0,Y 332.312,Z 538.734,A -85,B 0,C 180,E1 -14485.147,E2 -14485.147} C_VEL
LIN {X 0,Y 332.379,Z 539.808,A -85,B 0,C 180,E1 -14486.363,E2 -14486.363} C_VEL
LIN {X 0,Y 332.543,Z 540.417,A -85,B 0,C 180,E1 -14487.577,E2 -14487.577} C_VEL
LIN {X 0,Y 332.644,Z 540.597,A -85,B 0,C 180,E1 -14488.789,E2 -14488.789} C_VEL
LIN {X 0,Y 332.612,Z 540.344,A -85,B 0,C 180,E1 -14490,E2 -14490} C_VEL
LIN {X 0,Y 332.658,Z 539.612,A -85,B 0,C 180,E1 -14491.21,E2 -14491.21} C_VEL
LIN {X 0,Y 332.75,Z 538.448,A -85,B 0,C 180,E1 -14492.421,E2 -14492.421} C_VEL
LIN {X 0,Y 332.566,Z 535.763,A -85,B 0,C 180,E1 -14494.241,E2 -14494.241} C_VEL
LIN {X 0,Y 332.571,Z 531.949,A -85,B 0,C 180,E1 -14496.065,E2 -14496.065} C_VEL
LIN {X 0,Y 332.603,Z 526.828,A -85,B 0,C 180,E1 -14497.894,E2 -14497.894} C_VEL
LIN {X 0,Y 332.733,Z 520.219,A -85,B 0,C 180,E1 -14499.728,E2 -14499.728} C_VEL
LIN {X 0,Y 333.167,Z 511.895,A -85,B 0,C 180,E1 -14501.56,E2 -14501.56} C_VEL
LIN {X 0,Y 333.749,Z 503.206,A -85,B 0,C 180,E1 -14503.083,E2 -14503.083} C_VEL
LIN {X 0,Y 334.355,Z 493.588,A -85,B 0,C 180,E1 -14504.454,E2 -14504.454} C_VEL
LIN {X 0,Y 335.136,Z 482.813,A -85,B 0,C 180,E1 -14505.68,E2 -14505.68} C_VEL
LIN {X 0,Y 335.742,Z 472.992,A -85,B 0,C 180,E1 -14506.571,E2 -14506.571} C_VEL
LIN {X 0,Y 334.967,Z 460.437,A -85,B 0,C 180,E1 -14507.475,E2 -14507.475} C_VEL
LIN {X 0,Y 334.104,Z 448.062,A -85,B 0,C 180,E1 -14508.115,E2 -14508.115} C_VEL
LIN {X 0,Y 333.729,Z 440.601,A -85,B 0,C 180,E1 -14508.414,E2 -14508.414} C_VEL
LIN {X 0,Y 335.309,Z 426.125,A -85,B 0,C 180,E1 -14512.994,E2 -14512.994} C_VEL
LIN {X 0,Y 337.321,Z 411.685,A -85,B 0,C 180,E1 -14517.618,E2 -14517.618} C_VEL
LIN {X 0,Y 338.581,Z 403.626,A -85,B 0,C 180,E1 -14520.223,E2 -14520.223} C_VEL
LIN {X 0,Y 337.456,Z 397.29,A -85,B 0,C 180,E1 -14522.449,E2 -14522.449} C_VEL
LIN {X 0,Y 335.156,Z 386.135,A -85,B 0,C 180,E1 -14526.506,E2 -14526.506} C_VEL
LIN {X 0,Y 333.704,Z 378.917,A -85,B 0,C 180,E1 -14529.282,E2 -14529.282} C_VEL
LIN {X 0,Y 333.642,Z 378.926,A -85,B 0,C 180,E1 -14532.501,E2 -14532.501} C_VEL
LIN {X 0,Y 333.621,Z 378.928,A -85,B 0,C 180,E1 -14535.959,E2 -14535.959} C_VEL
LIN {X 0,Y 333.652,Z 378.921,A -85,B 0,C 180,E1 -14539.314,E2 -14539.314} C_VEL
LIN {X 0,Y 333.666,Z 378.919,A -85,B 0,C 180,E1 -14543.167,E2 -14543.167} C_VEL
LIN {X 0,Y 333.639,Z 378.923,A -85,B 0,C 180,E1 -14546.792,E2 -14546.792} C_VEL
LIN {X 0,Y 333.695,Z 378.919,A -85,B 0,C 180,E1 -14549.713,E2 -14549.713} C_VEL
LIN {X 0,Y 333.74,Z 378.912,A -85,B 0,C 180,E1 -14552.401,E2 -14552.401} C_VEL
LIN {X 0,Y 333.727,Z 378.912,A -85,B 0,C 180,E1 -14555.091,E2 -14555.091} C_VEL
LIN {X 0,Y 333.682,Z 378.917,A -85,B 0,C 180,E1 -14559.019,E2 -14559.019} C_VEL
LIN {X 0,Y 333.795,Z 378.907,A -85,B 0,C 180,E1 -14561.589,E2 -14561.589} C_VEL
LIN {X 0,Y 333.809,Z 378.906,A -85,B 0,C 180,E1 -14565.577,E2 -14565.577} C_VEL
LIN {X 0,Y 333.835,Z 378.899,A -85,B 0,C 180,E1 -14569.078,E2 -14569.078} C_VEL
LIN {X 0,Y 334.026,Z 378.874,A -85,B 0,C 180,E1 -14572.748,E2 -14572.748} C_VEL
LIN {X 0,Y 333.813,Z 378.903,A -85,B 0,C 180,E1 -14575.169,E2 -14575.169} C_VEL
LIN {X 0,Y 334.132,Z 378.866,A -85,B 0,C 180,E1 -14577.589,E2 -14577.589} C_VEL
LIN {X 0,Y 334.248,Z 378.848,A -85,B 0,C 180,E1 -14580,E2 -14580} C_VEL
LIN {X 0,Y 334.106,Z 378.864,A -85,B 0,C 180,E1 -14582.411,E2 -14582.411} C_VEL
LIN {X 0,Y 334.027,Z 378.879,A -85,B 0,C 180,E1 -14587.253,E2 -14587.253} C_VEL
LIN {X 0,Y 333.839,Z 378.9,A -85,B 0,C 180,E1 -14590.922,E2 -14590.922} C_VEL
LIN {X 0,Y 333.809,Z 378.902,A -85,B 0,C 180,E1 -14594.634,E2 -14594.634} C_VEL
LIN {X 0,Y 333.796,Z 378.904,A -85,B 0,C 180,E1 -14598.655,E2 -14598.655} C_VEL
LIN {X 0,Y 333.693,Z 378.916,A -85,B 0,C 180,E1 -14602.278,E2 -14602.278} C_VEL
LIN {X 0,Y 333.736,Z 378.91,A -85,B 0,C 180,E1 -14606.246,E2 -14606.246} C_VEL
LIN {X 0,Y 333.711,Z 378.919,A -85,B 0,C 180,E1 -14608.972,E2 -14608.972} C_VEL
LIN {X 0,Y 333.646,Z 378.924,A -85,B 0,C 180,E1 -14612.588,E2 -14612.588} C_VEL
LIN {X 0,Y 333.677,Z 378.918,A -85,B 0,C 180,E1 -14616.139,E2 -14616.139} C_VEL
LIN {X 0,Y 333.647,Z 378.924,A -85,B 0,C 180,E1 -14619.192,E2 -14619.192} C_VEL
LIN {X 0,Y 333.634,Z 378.926,A -85,B 0,C 180,E1 -14622.5,E2 -14622.5} C_VEL
LIN {X 0,Y 333.62,Z 378.925,A -85,B 0,C 180,E1 -14625.959,E2 -14625.959} C_VEL
LIN {X 0,Y 333.648,Z 378.922,A -85,B 0,C 180,E1 -14629.316,E2 -14629.316} C_VEL
LIN {X 0,Y 333.668,Z 378.92,A -85,B 0,C 180,E1 -14633.168,E2 -14633.168} C_VEL
LIN {X 0,Y 333.638,Z 378.926,A -85,B 0,C 180,E1 -14636.792,E2 -14636.792} C_VEL
LIN {X 0,Y 333.696,Z 378.916,A -85,B 0,C 180,E1 -14639.713,E2 -14639.713} C_VEL
LIN {X 0,Y 333.741,Z 378.915,A -85,B 0,C 180,E1 -14642.401,E2 -14642.401} C_VEL
LIN {X 0,Y 333.728,Z 378.912,A -85,B 0,C 180,E1 -14645.091,E2 -14645.091} C_VEL
LIN {X 0,Y 333.696,Z 378.916,A -85,B 0,C 180,E1 -14649.02,E2 -14649.02} C_VEL
LIN {X 0,Y 333.797,Z 378.903,A -85,B 0,C 180,E1 -14651.59,E2 -14651.59} C_VEL
LIN {X 0,Y 333.81,Z 378.902,A -85,B 0,C 180,E1 -14655.577,E2 -14655.577} C_VEL
LIN {X 0,Y 333.837,Z 378.898,A -85,B 0,C 180,E1 -14659.078,E2 -14659.078} C_VEL
LIN {X 0,Y 334.015,Z 378.876,A -85,B 0,C 180,E1 -14662.748,E2 -14662.748} C_VEL
LIN {X 0,Y 333.812,Z 378.901,A -85,B 0,C 180,E1 -14665.169,E2 -14665.169} C_VEL
LIN {X 0,Y 334.108,Z 378.866,A -85,B 0,C 180,E1 -14667.589,E2 -14667.589} C_VEL
LIN {X 0,Y 334.269,Z 378.85,A -85,B 0,C 180,E1 -14670,E2 -14670} C_VEL
LIN {X 0,Y 334.108,Z 378.866,A -85,B 0,C 180,E1 -14672.411,E2 -14672.411} C_VEL
LIN {X 0,Y 334.017,Z 378.88,A -85,B 0,C 180,E1 -14676.039,E2 -14676.039} C_VEL
LIN {X 0,Y 333.961,Z 378.883,A -85,B 0,C 180,E1 -14678.471,E2 -14678.471} C_VEL
LIN {X 0,Y 333.794,Z 378.906,A -85,B 0,C 180,E1 -14682.155,E2 -14682.155} C_VEL
LIN {X 0,Y 333.781,Z 378.909,A -85,B 0,C 180,E1 -14685.886,E2 -14685.886} C_VEL
LIN {X 0,Y 333.8,Z 378.903,A -85,B 0,C 180,E1 -14688.656,E2 -14688.656} C_VEL
LIN {X 0,Y 333.695,Z 378.916,A -85,B 0,C 180,E1 -14692.278,E2 -14692.278} C_VEL
LIN {X 0,Y 333.738,Z 378.911,A -85,B 0,C 180,E1 -14696.246,E2 -14696.246} C_VEL
LIN {X 0,Y 333.693,Z 378.917,A -85,B 0,C 180,E1 -14698.974,E2 -14698.974} C_VEL
LIN {X 0,Y 333.646,Z 378.922,A -85,B 0,C 180,E1 -14702.587,E2 -14702.587} C_VEL
LIN {X 0,Y 333.679,Z 378.918,A -85,B 0,C 180,E1 -14706.139,E2 -14706.139} C_VEL
LIN {X 0,Y 333.65,Z 378.926,A -85,B 0,C 180,E1 -14709.192,E2 -14709.192} C_VEL
LIN {X 0,Y 333.635,Z 378.923,A -85,B 0,C 180,E1 -14712.5,E2 -14712.5} C_VEL
LIN {X 0,Y 333.625,Z 378.925,A -85,B 0,C 180,E1 -14715.959,E2 -14715.959} C_VEL
LIN {X 0,Y 333.65,Z 378.926,A -85,B 0,C 180,E1 -14719.315,E2 -14719.315} C_VEL
LIN {X 0,Y 333.668,Z 378.924,A -85,B 0,C 180,E1 -14723.168,E2 -14723.168} C_VEL
LIN {X 0,Y 333.687,Z 378.92,A -85,B 0,C 180,E1 -14726.797,E2 -14726.797} C_VEL
LIN {X 0,Y 333.875,Z 378.972,A -85,B 0,C 180,E1 -14728.443,E2 -14728.443} C_VEL
LIN {X 0,Y 333.995,Z 382.014,A -85,B 0,C 180,E1 -14730.364,E2 -14730.364} C_VEL
LIN {X 0,Y 333.64,Z 387.555,A -85,B 0,C 180,E1 -14733.745,E2 -14733.745} C_VEL
LIN {X 0,Y 333.278,Z 394.084,A -85,B 0,C 180,E1 -14737.693,E2 -14737.693} C_VEL
LIN {X 0,Y 333.137,Z 396.949,A -85,B 0,C 180,E1 -14739.398,E2 -14739.398} C_VEL
LIN {X 0,Y 332.437,Z 398.65,A -85,B 0,C 180,E1 -14740.363,E2 -14740.363} C_VEL
LIN {X 0,Y 329.477,Z 401.583,A -85,B 0,C 180,E1 -14741.921,E2 -14741.921} C_VEL
LIN {X 0,Y 326.951,Z 403.973,A -85,B 0,C 180,E1 -14743.181,E2 -14743.181} C_VEL
LIN {X 0,Y 325.834,Z 405.74,A -85,B 0,C 180,E1 -14744.161,E2 -14744.161} C_VEL
LIN {X 0,Y 325.726,Z 406.324,A -85,B 0,C 180,E1 -14744.494,E2 -14744.494} C_VEL
LIN {X 0,Y 325.563,Z 412.156,A -85,B 0,C 180,E1 -14747.85,E2 -14747.85} C_VEL
LIN {X 0,Y 326.784,Z 423.846,A -85,B 0,C 180,E1 -14748.682,E2 -14748.682} C_VEL
LIN {X 0,Y 327.519,Z 431.167,A -85,B 0,C 180,E1 -14749.334,E2 -14749.334} C_VEL
LIN {X 0,Y 326.997,Z 441.128,A -85,B 0,C 180,E1 -14750.412,E2 -14750.412} C_VEL
LIN {X 0,Y 326.627,Z 449.877,A -85,B 0,C 180,E1 -14751.614,E2 -14751.614} C_VEL
LIN {X 0,Y 326.368,Z 457.319,A -85,B 0,C 180,E1 -14752.887,E2 -14752.887} C_VEL
LIN {X 0,Y 326.072,Z 464.513,A -85,B 0,C 180,E1 -14754.434,E2 -14754.434} C_VEL
LIN {X 0,Y 325.902,Z 469.108,A -85,B 0,C 180,E1 -14755.671,E2 -14755.671} C_VEL
LIN {X 0,Y 325.653,Z 472.833,A -85,B 0,C 180,E1 -14756.907,E2 -14756.907} C_VEL
LIN {X 0,Y 325.516,Z 476.94,A -85,B 0,C 180,E1 -14758.763,E2 -14758.763} C_VEL
LIN {X 0,Y 325.565,Z 478.803,A -85,B 0,C 180,E1 -14760,E2 -14760} C_VEL
LIN {X 0,Y 325.689,Z 480.009,A -85,B 0,C 180,E1 -14761.236,E2 -14761.236} C_VEL
LIN {X 0,Y 325.88,Z 480.575,A -85,B 0,C 180,E1 -14762.472,E2 -14762.472} C_VEL
LIN {X 0,Y 326.221,Z 480.499,A -85,B 0,C 180,E1 -14763.706,E2 -14763.706} C_VEL
LIN {X 0,Y 326.774,Z 479.774,A -85,B 0,C 180,E1 -14764.935,E2 -14764.935} C_VEL
LIN {X 0,Y 327.4,Z 478.437,A -85,B 0,C 180,E1 -14766.161,E2 -14766.161} C_VEL
LIN {X 0,Y 328.606,Z 475.177,A -85,B 0,C 180,E1 -14767.991,E2 -14767.991} C_VEL
LIN {X 0,Y 329.89,Z 470.338,A -85,B 0,C 180,E1 -14769.813,E2 -14769.813} C_VEL
LIN {X 0,Y 331.557,Z 463.628,A -85,B 0,C 180,E1 -14771.617,E2 -14771.617} C_VEL
LIN {X 0,Y 333.16,Z 456.413,A -85,B 0,C 180,E1 -14773.107,E2 -14773.107} C_VEL
LIN {X 0,Y 334.765,Z 448.301,A -85,B 0,C 180,E1 -14774.423,E2 -14774.423} C_VEL
LIN {X 0,Y 335.062,Z 445.222,A -85,B 0,C 180,E1 -14774.88,E2 -14774.88} C_VEL
LIN {X 0,Y 334.093,Z 437.602,A -85,B 0,C 180,E1 -14776.081,E2 -14776.081} C_VEL
LIN {X 0,Y 331.657,Z 428.076,A -85,B 0,C 180,E1 -14777.526,E2 -14777.526} C_VEL
LIN {X 0,Y 328.417,Z 418.643,A -85,B 0,C 180,E1 -14778.92,E2 -14778.92} C_VEL
LIN {X 0,Y 329.195,Z 414.231,A -85,B 0,C 180,E1 -14782.599,E2 -14782.599} C_VEL
LIN {X 0,Y 330.311,Z 409.884,A -85,B 0,C 180,E1 -14786.666,E2 -14786.666} C_VEL
LIN {X 0,Y 331.172,Z 407.242,A -85,B 0,C 180,E1 -14789.531,E2 -14789.531} C_VEL
LIN {X 0,Y 331.695,Z 405.331,A -85,B 0,C 180,E1 -14792.056,E2 -14792.056} C_VEL
LIN {X 0,Y 331.872,Z 403.831,A -85,B 0,C 180,E1 -14794.874,E2 -14794.874} C_VEL
LIN {X 0,Y 331.996,Z 402.864,A -85,B 0,C 180,E1 -14797.872,E2 -14797.872} C_VEL
LIN {X 0,Y 332.165,Z 402.666,A -85,B 0,C 180,E1 -14800.988,E2 -14800.988} C_VEL
LIN {X 0,Y 332.489,Z 403.343,A -85,B 0,C 180,E1 -14804.23,E2 -14804.23} C_VEL
LIN {X 0,Y 332.983,Z 405.125,A -85,B 0,C 180,E1 -14807.622,E2 -14807.622} C_VEL
LIN {X 0,Y 333.316,Z 406.501,A -85,B 0,C 180,E1 -14809.382,E2 -14809.382} C_VEL
LIN {X 0,Y 334.171,Z 410.415,A -85,B 0,C 180,E1 -14813.052,E2 -14813.052} C_VEL
LIN {X 0,Y 335.007,Z 413.774,A -85,B 0,C 180,E1 -14815.498,E2 -14815.498} C_VEL
LIN {X 0,Y 335.527,Z 417.466,A -85,B 0,C 180,E1 -14817.715,E2 -14817.715} C_VEL
LIN {X 0,Y 335.233,Z 420.056,A -85,B 0,C 180,E1 -14819.004,E2 -14819.004} C_VEL
LIN {X 0,Y 332.431,Z 428.755,A -85,B 0,C 180,E1 -14822.615,E2 -14822.615} C_VEL
LIN {X 0,Y 330.265,Z 437.511,A -85,B 0,C 180,E1 -14825.926,E2 -14825.926} C_VEL
LIN {X 0,Y 333.256,Z 451.505,A -85,B 0,C 180,E1 -14827.136,E2 -14827.136} C_VEL
LIN {X 0,Y 334.463,Z 462.048,A -85,B 0,C 180,E1 -14828.094,E2 -14828.094} C_VEL
LIN {X 0,Y 334.489,Z 472.209,A -85,B 0,C 180,E1 -14829.072,E2 -14829.072} C_VEL
LIN {X 0,Y 333.567,Z 482.134,A -85,B 0,C 180,E1 -14830.139,E2 -14830.139} C_VEL
LIN {X 0,Y 331.7,Z 492.788,A -85,B 0,C 180,E1 -14831.469,E2 -14831.469} C_VEL
LIN {X 0,Y 329.955,Z 502.391,A -85,B 0,C 180,E1 -14832.97,E2 -14832.97} C_VEL
LIN {X 0,Y 328.212,Z 511.924,A -85,B 0,C 180,E1 -14834.816,E2 -14834.816} C_VEL
LIN {X 0,Y 326.999,Z 519.413,A -85,B 0,C 180,E1 -14836.641,E2 -14836.641} C_VEL
LIN {X 0,Y 325.867,Z 526.501,A -85,B 0,C 180,E1 -14838.807,E2 -14838.807} C_VEL
LIN {X 0,Y 325.426,Z 531.237,A -85,B 0,C 180,E1 -14840.678,E2 -14840.678} C_VEL
LIN {X 0,Y 325.274,Z 534.875,A -85,B 0,C 180,E1 -14842.551,E2 -14842.551} C_VEL
LIN {X 0,Y 325.233,Z 536.723,A -85,B 0,C 180,E1 -14843.797,E2 -14843.797} C_VEL
LIN {X 0,Y 325.244,Z 538.158,A -85,B 0,C 180,E1 -14845.041,E2 -14845.041} C_VEL
LIN {X 0,Y 325.293,Z 539.138,A -85,B 0,C 180,E1 -14846.283,E2 -14846.283} C_VEL
LIN {X 0,Y 325.473,Z 539.692,A -85,B 0,C 180,E1 -14847.525,E2 -14847.525} C_VEL
LIN {X 0,Y 325.597,Z 539.827,A -85,B 0,C 180,E1 -14848.763,E2 -14848.763} C_VEL
LIN {X 0,Y 325.569,Z 539.483,A -85,B 0,C 180,E1 -14850,E2 -14850} C_VEL
LIN {X 0,Y 325.617,Z 538.693,A -85,B 0,C 180,E1 -14851.237,E2 -14851.237} C_VEL
LIN {X 0,Y 325.705,Z 537.481,A -85,B 0,C 180,E1 -14852.473,E2 -14852.473} C_VEL
LIN {X 0,Y 325.523,Z 534.681,A -85,B 0,C 180,E1 -14854.333,E2 -14854.333} C_VEL
LIN {X 0,Y 325.519,Z 530.714,A -85,B 0,C 180,E1 -14856.197,E2 -14856.197} C_VEL
LIN {X 0,Y 325.549,Z 525.428,A -85,B 0,C 180,E1 -14858.066,E2 -14858.066} C_VEL
LIN {X 0,Y 325.701,Z 518.66,A -85,B 0,C 180,E1 -14859.94,E2 -14859.94} C_VEL
LIN {X 0,Y 326.087,Z 511.663,A -85,B 0,C 180,E1 -14861.499,E2 -14861.499} C_VEL
LIN {X 0,Y 326.653,Z 503.058,A -85,B 0,C 180,E1 -14863.056,E2 -14863.056} C_VEL
LIN {X 0,Y 327.245,Z 493.54,A -85,B 0,C 180,E1 -14864.457,E2 -14864.457} C_VEL
LIN {X 0,Y 328.055,Z 483.087,A -85,B 0,C 180,E1 -14865.696,E2 -14865.696} C_VEL
LIN {X 0,Y 328.652,Z 473.327,A -85,B 0,C 180,E1 -14866.619,E2 -14866.619} C_VEL
LIN {X 0,Y 327.898,Z 461.017,A -85,B 0,C 180,E1 -14867.542,E2 -14867.542} C_VEL
LIN {X 0,Y 327.044,Z 448.276,A -85,B 0,C 180,E1 -14868.236,E2 -14868.236} C_VEL
LIN {X 0,Y 326.69,Z 440.267,A -85,B 0,C 180,E1 -14868.582,E2 -14868.582} C_VEL
LIN {X 0,Y 328.371,Z 425.549,A -85,B 0,C 180,E1 -14873.39,E2 -14873.39} C_VEL
LIN {X 0,Y 330.383,Z 411.835,A -85,B 0,C 180,E1 -14877.904,E2 -14877.904} C_VEL
LIN {X 0,Y 331.499,Z 405.514,A -85,B 0,C 180,E1 -14879.992,E2 -14879.992} C_VEL
LIN {X 0,Y 331.238,Z 402.034,A -85,B 0,C 180,E1 -14881.193,E2 -14881.193} C_VEL
LIN {X 0,Y 328.933,Z 391.09,A -85,B 0,C 180,E1 -14885.231,E2 -14885.231} C_VEL
LIN {X 0,Y 327.183,Z 382.517,A -85,B 0,C 180,E1 -14888.53,E2 -14888.53} C_VEL
LIN {X 0,Y 326.626,Z 379.799,A -85,B 0,C 180,E1 -14889.671,E2 -14889.671} C_VEL
LIN {X 0,Y 326.587,Z 379.801,A -85,B 0,C 180,E1 -14893.521,E2 -14893.521} C_VEL
LIN {X 0,Y 326.584,Z 379.801,A -85,B 0,C 180,E1 -14897.026,E2 -14897.026} C_VEL
LIN {X 0,Y 326.615,Z 379.798,A -85,B 0,C 180,E1 -14900.772,E2 -14900.772} C_VEL
LIN {X 0,Y 326.613,Z 379.8,A -85,B 0,C 180,E1 -14904.48,E2 -14904.48} C_VEL
LIN {X 0,Y 326.61,Z 379.799,A -85,B 0,C 180,E1 -14907.456,E2 -14907.456} C_VEL
LIN {X 0,Y 326.648,Z 379.796,A -85,B 0,C 180,E1 -14910.34,E2 -14910.34} C_VEL
LIN {X 0,Y 326.69,Z 379.789,A -85,B 0,C 180,E1 -14914.516,E2 -14914.516} C_VEL
LIN {X 0,Y 326.647,Z 379.794,A -85,B 0,C 180,E1 -14918.545,E2 -14918.545} C_VEL
LIN {X 0,Y 326.745,Z 379.782,A -85,B 0,C 180,E1 -14921.177,E2 -14921.177} C_VEL
LIN {X 0,Y 326.764,Z 379.782,A -85,B 0,C 180,E1 -14925.433,E2 -14925.433} C_VEL
LIN {X 0,Y 326.771,Z 379.778,A -85,B 0,C 180,E1 -14928.839,E2 -14928.839} C_VEL
LIN {X 0,Y 326.98,Z 379.752,A -85,B 0,C 180,E1 -14932.59,E2 -14932.59} C_VEL
LIN {X 0,Y 326.78,Z 379.778,A -85,B 0,C 180,E1 -14935.065,E2 -14935.065} C_VEL
LIN {X 0,Y 327.069,Z 379.747,A -85,B 0,C 180,E1 -14937.537,E2 -14937.537} C_VEL
LIN {X 0,Y 327.2,Z 379.726,A -85,B 0,C 180,E1 -14940,E2 -14940} C_VEL
LIN {X 0,Y 327.047,Z 379.743,A -85,B 0,C 180,E1 -14942.463,E2 -14942.463} C_VEL
LIN {X 0,Y 326.972,Z 379.753,A -85,B 0,C 180,E1 -14946.672,E2 -14946.672} C_VEL
LIN {X 0,Y 326.816,Z 379.773,A -85,B 0,C 180,E1 -14949.906,E2 -14949.906} C_VEL
LIN {X 0,Y 326.761,Z 379.781,A -85,B 0,C 180,E1 -14953.685,E2 -14953.685} C_VEL
LIN {X 0,Y 326.7,Z 379.789,A -85,B 0,C 180,E1 -14957.528,E2 -14957.528} C_VEL
LIN {X 0,Y 326.666,Z 379.791,A -85,B 0,C 180,E1 -14960.135,E2 -14960.135} C_VEL
LIN {X 0,Y 326.653,Z 379.793,A -85,B 0,C 180,E1 -14964.129,E2 -14964.129} C_VEL
LIN {X 0,Y 326.685,Z 379.792,A -85,B 0,C 180,E1 -14966.858,E2 -14966.858} C_VEL
LIN {X 0,Y 326.639,Z 379.797,A -85,B 0,C 180,E1 -14970.611,E2 -14970.611} C_VEL
LIN {X 0,Y 326.608,Z 379.798,A -85,B 0,C 180,E1 -14974.019,E2 -14974.019} C_VEL
LIN {X 0,Y 326.629,Z 379.798,A -85,B 0,C 180,E1 -14977.239,E2 -14977.239} C_VEL
LIN {X 0,Y 326.578,Z 379.805,A -85,B 0,C 180,E1 -14981.132,E2 -14981.132} C_VEL
LIN {X 0,Y 326.558,Z 379.81,A -85,B 0,C 180,E1 -14984.748,E2 -14984.748} C_VEL
LIN {X 0,Y 326.577,Z 379.803,A -85,B 0,C 180,E1 -14988.155,E2 -14988.155} C_VEL
LIN {X 0,Y 326.625,Z 379.796,A -85,B 0,C 180,E1 -14991.392,E2 -14991.392} C_VEL
LIN {X 0,Y 326.621,Z 379.8,A -85,B 0,C 180,E1 -14994.851,E2 -14994.851} C_VEL
LIN {X 0,Y 326.609,Z 379.798,A -85,B 0,C 180,E1 -14997.456,E2 -14997.456} C_VEL
LIN {X 0,Y 326.649,Z 379.797,A -85,B 0,C 180,E1 -15000.34,E2 -15000.34} C_VEL
LIN {X 0,Y 326.691,Z 379.793,A -85,B 0,C 180,E1 -15004.517,E2 -15004.517} C_VEL
LIN {X 0,Y 326.655,Z 379.796,A -85,B 0,C 180,E1 -15008.546,E2 -15008.546} C_VEL
LIN {X 0,Y 326.746,Z 379.781,A -85,B 0,C 180,E1 -15011.178,E2 -15011.178} C_VEL
LIN {X 0,Y 326.765,Z 379.779,A -85,B 0,C 180,E1 -15015.433,E2 -15015.433} C_VEL
LIN {X 0,Y 326.773,Z 379.778,A -85,B 0,C 180,E1 -15018.839,E2 -15018.839} C_VEL
LIN {X 0,Y 326.968,Z 379.755,A -85,B 0,C 180,E1 -15022.59,E2 -15022.59} C_VEL
LIN {X 0,Y 326.779,Z 379.777,A -85,B 0,C 180,E1 -15025.065,E2 -15025.065} C_VEL
LIN {X 0,Y 327.049,Z 379.745,A -85,B 0,C 180,E1 -15027.537,E2 -15027.537} C_VEL
LIN {X 0,Y 327.22,Z 379.728,A -85,B 0,C 180,E1 -15030,E2 -15030} C_VEL
LIN {X 0,Y 327.049,Z 379.745,A -85,B 0,C 180,E1 -15032.463,E2 -15032.463} C_VEL
LIN {X 0,Y 326.991,Z 379.754,A -85,B 0,C 180,E1 -15036.169,E2 -15036.169} C_VEL
LIN {X 0,Y 326.809,Z 379.778,A -85,B 0,C 180,E1 -15039.907,E2 -15039.907} C_VEL
LIN {X 0,Y 326.762,Z 379.784,A -85,B 0,C 180,E1 -15043.686,E2 -15043.686} C_VEL
LIN {X 0,Y 326.703,Z 379.79,A -85,B 0,C 180,E1 -15047.528,E2 -15047.528} C_VEL
LIN {X 0,Y 326.668,Z 379.792,A -85,B 0,C 180,E1 -15050.135,E2 -15050.135} C_VEL
LIN {X 0,Y 326.655,Z 379.794,A -85,B 0,C 180,E1 -15054.129,E2 -15054.129} C_VEL
LIN {X 0,Y 326.685,Z 379.789,A -85,B 0,C 180,E1 -15056.858,E2 -15056.858} C_VEL
LIN {X 0,Y 326.636,Z 379.795,A -85,B 0,C 180,E1 -15060.61,E2 -15060.61} C_VEL
LIN {X 0,Y 326.609,Z 379.799,A -85,B 0,C 180,E1 -15064.019,E2 -15064.019} C_VEL
LIN {X 0,Y 326.632,Z 379.8,A -85,B 0,C 180,E1 -15067.239,E2 -15067.239} C_VEL
LIN {X 0,Y 326.581,Z 379.806,A -85,B 0,C 180,E1 -15071.132,E2 -15071.132} C_VEL
LIN {X 0,Y 326.558,Z 379.806,A -85,B 0,C 180,E1 -15074.748,E2 -15074.748} C_VEL
LIN {X 0,Y 326.579,Z 379.802,A -85,B 0,C 180,E1 -15078.154,E2 -15078.154} C_VEL
LIN {X 0,Y 326.626,Z 379.799,A -85,B 0,C 180,E1 -15081.392,E2 -15081.392} C_VEL
LIN {X 0,Y 326.628,Z 379.799,A -85,B 0,C 180,E1 -15084.85,E2 -15084.85} C_VEL
LIN {X 0,Y 326.832,Z 379.869,A -85,B 0,C 180,E1 -15088.389,E2 -15088.389} C_VEL
LIN {X 0,Y 326.878,Z 384.072,A -85,B 0,C 180,E1 -15091.069,E2 -15091.069} C_VEL
LIN {X 0,Y 326.477,Z 389.929,A -85,B 0,C 180,E1 -15094.707,E2 -15094.707} C_VEL
LIN {X 0,Y 326.137,Z 396.201,A -85,B 0,C 180,E1 -15098.51,E2 -15098.51} C_VEL
LIN {X 0,Y 325.888,Z 402.783,A -85,B 0,C 180,E1 -15102.427,E2 -15102.427} C_VEL
LIN {X 0,Y 325.726,Z 406.324,A -85,B 0,C 180,E1 -15104.494,E2 -15104.494} C_VEL
LIN {X 0,Y 325.013,Z 408.255,A -85,B 0,C 180,E1 -15105.425,E2 -15105.425} C_VEL
LIN {X 0,Y 322.861,Z 411.645,A -85,B 0,C 180,E1 -15106.57,E2 -15106.57} C_VEL
LIN {X 0,Y 320.62,Z 416.077,A -85,B 0,C 180,E1 -15107.571,E2 -15107.571} C_VEL
LIN {X 0,Y 319.615,Z 420.245,A -85,B 0,C 180,E1 -15108.198,E2 -15108.198} C_VEL
LIN {X 0,Y 319.606,Z 423.429,A -85,B 0,C 180,E1 -15108.523,E2 -15108.523} C_VEL
LIN {X 0,Y 320.433,Z 431.551,A -85,B 0,C 180,E1 -15109.255,E2 -15109.255} C_VEL
LIN {X 0,Y 319.915,Z 441.545,A -85,B 0,C 180,E1 -15110.357,E2 -15110.357} C_VEL
LIN {X 0,Y 319.521,Z 450.897,A -85,B 0,C 180,E1 -15111.673,E2 -15111.673} C_VEL
LIN {X 0,Y 319.257,Z 458.637,A -85,B 0,C 180,E1 -15113.046,E2 -15113.046} C_VEL
LIN {X 0,Y 318.949,Z 465.665,A -85,B 0,C 180,E1 -15114.626,E2 -15114.626} C_VEL
LIN {X 0,Y 318.599,Z 471.135,A -85,B 0,C 180,E1 -15116.206,E2 -15116.206} C_VEL
LIN {X 0,Y 318.443,Z 476.018,A -85,B 0,C 180,E1 -15118.103,E2 -15118.103} C_VEL
LIN {X 0,Y 318.49,Z 479.28,A -85,B 0,C 180,E1 -15120,E2 -15120} C_VEL
LIN {X 0,Y 318.646,Z 480.622,A -85,B 0,C 180,E1 -15121.264,E2 -15121.264} C_VEL
LIN {X 0,Y 318.844,Z 481.327,A -85,B 0,C 180,E1 -15122.527,E2 -15122.527} C_VEL
LIN {X 0,Y 319.196,Z 481.395,A -85,B 0,C 180,E1 -15123.787,E2 -15123.787} C_VEL
LIN {X 0,Y 319.776,Z 480.812,A -85,B 0,C 180,E1 -15125.043,E2 -15125.043} C_VEL
LIN {X 0,Y 320.436,Z 479.599,A -85,B 0,C 180,E1 -15126.296,E2 -15126.296} C_VEL
LIN {X 0,Y 321.702,Z 476.549,A -85,B 0,C 180,E1 -15128.164,E2 -15128.164} C_VEL
LIN {X 0,Y 323.077,Z 471.999,A -85,B 0,C 180,E1 -15130.022,E2 -15130.022} C_VEL
LIN {X 0,Y 324.534,Z 466.877,A -85,B 0,C 180,E1 -15131.555,E2 -15131.555} C_VEL
LIN {X 0,Y 326.161,Z 460.333,A -85,B 0,C 180,E1 -15133.076,E2 -15133.076} C_VEL
LIN {X 0,Y 328.041,Z 452.094,A -85,B 0,C 180,E1 -15134.56,E2 -15134.56} C_VEL
LIN {X 0,Y 328.736,Z 447.748,A -85,B 0,C 180,E1 -15135.249,E2 -15135.249} C_VEL
LIN {X 0,Y 327.943,Z 440.126,A -85,B 0,C 180,E1 -15136.534,E2 -15136.534} C_VEL
LIN {X 0,Y 325.468,Z 430.059,A -85,B 0,C 180,E1 -15138.173,E2 -15138.173} C_VEL
LIN {X 0,Y 321.757,Z 419.293,A -85,B 0,C 180,E1 -15139.879,E2 -15139.879} C_VEL
LIN {X 0,Y 322.794,Z 414.215,A -85,B 0,C 180,E1 -15144.436,E2 -15144.436} C_VEL
LIN {X 0,Y 323.623,Z 411.536,A -85,B 0,C 180,E1 -15147.133,E2 -15147.133} C_VEL
LIN {X 0,Y 324.481,Z 409.089,A -85,B 0,C 180,E1 -15149.96,E2 -15149.96} C_VEL
LIN {X 0,Y 325.019,Z 407.229,A -85,B 0,C 180,E1 -15152.723,E2 -15152.723} C_VEL
LIN {X 0,Y 325.191,Z 405.89,A -85,B 0,C 180,E1 -15155.699,E2 -15155.699} C_VEL
LIN {X 0,Y 325.386,Z 405.21,A -85,B 0,C 180,E1 -15158.961,E2 -15158.961} C_VEL
LIN {X 0,Y 325.607,Z 405.336,A -85,B 0,C 180,E1 -15161.999,E2 -15161.999} C_VEL
LIN {X 0,Y 325.896,Z 406.053,A -85,B 0,C 180,E1 -15164.63,E2 -15164.63} C_VEL
LIN {X 0,Y 326.429,Z 408.068,A -85,B 0,C 180,E1 -15168.131,E2 -15168.131} C_VEL
LIN {X 0,Y 327.092,Z 411.083,A -85,B 0,C 180,E1 -15171.457,E2 -15171.457} C_VEL
LIN {X 0,Y 328.045,Z 415,A -85,B 0,C 180,E1 -15174.658,E2 -15174.658} C_VEL
LIN {X 0,Y 328.721,Z 418.767,A -85,B 0,C 180,E1 -15177.115,E2 -15177.115} C_VEL
LIN {X 0,Y 328.664,Z 421.144,A -85,B 0,C 180,E1 -15178.406,E2 -15178.406} C_VEL
LIN {X 0,Y 327.176,Z 425.591,A -85,B 0,C 180,E1 -15180.392,E2 -15180.392} C_VEL
LIN {X 0,Y 324.287,Z 435.227,A -85,B 0,C 180,E1 -15184.313,E2 -15184.313} C_VEL
LIN {X 0,Y 323.856,Z 437.237,A -85,B 0,C 180,E1 -15185.05,E2 -15185.05} C_VEL
LIN {X 0,Y 326.713,Z 450.106,A -85,B 0,C 180,E1 -15186.245,E2 -15186.245} C_VEL
LIN {X 0,Y 328.124,Z 461.235,A -85,B 0,C 180,E1 -15187.323,E2 -15187.323} C_VEL
LIN {X 0,Y 328.256,Z 471.071,A -85,B 0,C 180,E1 -15188.32,E2 -15188.32} C_VEL
LIN {X 0,Y 327.216,Z 482.243,A -85,B 0,C 180,E1 -15189.572,E2 -15189.572} C_VEL
LIN {X 0,Y 325.247,Z 492.672,A -85,B 0,C 180,E1 -15190.924,E2 -15190.924} C_VEL
LIN {X 0,Y 323.212,Z 502.963,A -85,B 0,C 180,E1 -15192.603,E2 -15192.603} C_VEL
LIN {X 0,Y 321.513,Z 511.373,A -85,B 0,C 180,E1 -15194.3,E2 -15194.3} C_VEL
LIN {X 0,Y 320.084,Z 519.455,A -85,B 0,C 180,E1 -15196.347,E2 -15196.347} C_VEL
LIN {X 0,Y 319.178,Z 524.522,A -85,B 0,C 180,E1 -15197.925,E2 -15197.925} C_VEL
LIN {X 0,Y 318.502,Z 529.499,A -85,B 0,C 180,E1 -15199.832,E2 -15199.832} C_VEL
LIN {X 0,Y 318.197,Z 533.363,A -85,B 0,C 180,E1 -15201.746,E2 -15201.746} C_VEL
LIN {X 0,Y 318.151,Z 536.33,A -85,B 0,C 180,E1 -15203.752,E2 -15203.752} C_VEL
LIN {X 0,Y 318.179,Z 537.564,A -85,B 0,C 180,E1 -15204.931,E2 -15204.931} C_VEL
LIN {X 0,Y 318.403,Z 538.964,A -85,B 0,C 180,E1 -15207.47,E2 -15207.47} C_VEL
LIN {X 0,Y 318.551,Z 539.028,A -85,B 0,C 180,E1 -15208.736,E2 -15208.736} C_VEL
LIN {X 0,Y 318.527,Z 538.6,A -85,B 0,C 180,E1 -15210,E2 -15210} C_VEL
LIN {X 0,Y 318.577,Z 537.762,A -85,B 0,C 180,E1 -15211.264,E2 -15211.264} C_VEL
LIN {X 0,Y 318.66,Z 536.458,A -85,B 0,C 180,E1 -15212.528,E2 -15212.528} C_VEL
LIN {X 0,Y 318.483,Z 533.521,A -85,B 0,C 180,E1 -15214.429,E2 -15214.429} C_VEL
LIN {X 0,Y 318.464,Z 529.408,A -85,B 0,C 180,E1 -15216.335,E2 -15216.335} C_VEL
LIN {X 0,Y 318.516,Z 523.979,A -85,B 0,C 180,E1 -15218.246,E2 -15218.246} C_VEL
LIN {X 0,Y 318.698,Z 516.999,A -85,B 0,C 180,E1 -15220.161,E2 -15220.161} C_VEL
LIN {X 0,Y 319.194,Z 508.153,A -85,B 0,C 180,E1 -15222.074,E2 -15222.074} C_VEL
LIN {X 0,Y 319.769,Z 498.885,A -85,B 0,C 180,E1 -15223.666,E2 -15223.666} C_VEL
LIN {X 0,Y 320.588,Z 488.373,A -85,B 0,C 180,E1 -15225.116,E2 -15225.116} C_VEL
LIN {X 0,Y 321.359,Z 477.12,A -85,B 0,C 180,E1 -15226.337,E2 -15226.337} C_VEL
LIN {X 0,Y 321.43,Z 470.586,A -85,B 0,C 180,E1 -15226.922,E2 -15226.922} C_VEL
LIN {X 0,Y 320.649,Z 458.81,A -85,B 0,C 180,E1 -15227.787,E2 -15227.787} C_VEL
LIN {X 0,Y 319.835,Z 445.597,A -85,B 0,C 180,E1 -15228.481,E2 -15228.481} C_VEL
LIN {X 0,Y 319.62,Z 440.036,A -85,B 0,C 180,E1 -15228.72,E2 -15228.72} C_VEL
LIN {X 0,Y 321.212,Z 426.62,A -85,B 0,C 180,E1 -15233.227,E2 -15233.227} C_VEL
LIN {X 0,Y 323.278,Z 412.882,A -85,B 0,C 180,E1 -15237.866,E2 -15237.866} C_VEL
LIN {X 0,Y 324.368,Z 406.846,A -85,B 0,C 180,E1 -15239.926,E2 -15239.926} C_VEL
LIN {X 0,Y 324.362,Z 403.901,A -85,B 0,C 180,E1 -15240.97,E2 -15240.97} C_VEL
LIN {X 0,Y 322.359,Z 394.34,A -85,B 0,C 180,E1 -15244.53,E2 -15244.53} C_VEL
LIN {X 0,Y 320.42,Z 384.751,A -85,B 0,C 180,E1 -15248.288,E2 -15248.288} C_VEL
LIN {X 0,Y 319.588,Z 380.677,A -85,B 0,C 180,E1 -15249.976,E2 -15249.976} C_VEL
LIN {X 0,Y 319.567,Z 380.676,A -85,B 0,C 180,E1 -15253.469,E2 -15253.469} C_VEL
LIN {X 0,Y 319.562,Z 380.676,A -85,B 0,C 180,E1 -15257.018,E2 -15257.018} C_VEL
LIN {X 0,Y 319.551,Z 380.681,A -85,B 0,C 180,E1 -15260.371,E2 -15260.371} C_VEL
LIN {X 0,Y 319.56,Z 380.677,A -85,B 0,C 180,E1 -15263.572,E2 -15263.572} C_VEL
LIN {X 0,Y 319.578,Z 380.675,A -85,B 0,C 180,E1 -15266.686,E2 -15266.686} C_VEL
LIN {X 0,Y 319.585,Z 380.675,A -85,B 0,C 180,E1 -15269.616,E2 -15269.616} C_VEL
LIN {X 0,Y 319.606,Z 380.672,A -85,B 0,C 180,E1 -15272.498,E2 -15272.498} C_VEL
LIN {X 0,Y 319.605,Z 380.671,A -85,B 0,C 180,E1 -15275.304,E2 -15275.304} C_VEL
LIN {X 0,Y 319.597,Z 380.675,A -85,B 0,C 180,E1 -15278.048,E2 -15278.048} C_VEL
LIN {X 0,Y 319.69,Z 380.66,A -85,B 0,C 180,E1 -15280.962,E2 -15280.962} C_VEL
LIN {X 0,Y 319.731,Z 380.656,A -85,B 0,C 180,E1 -15285.276,E2 -15285.276} C_VEL
LIN {X 0,Y 319.759,Z 380.655,A -85,B 0,C 180,E1 -15289.873,E2 -15289.873} C_VEL
LIN {X 0,Y 319.934,Z 380.63,A -85,B 0,C 180,E1 -15292.426,E2 -15292.426} C_VEL
LIN {X 0,Y 319.749,Z 380.653,A -85,B 0,C 180,E1 -15294.956,E2 -15294.956} C_VEL
LIN {X 0,Y 320.01,Z 380.625,A -85,B 0,C 180,E1 -15297.483,E2 -15297.483} C_VEL
LIN {X 0,Y 320.152,Z 380.604,A -85,B 0,C 180,E1 -15300,E2 -15300} C_VEL
LIN {X 0,Y 319.991,Z 380.622,A -85,B 0,C 180,E1 -15302.518,E2 -15302.518} C_VEL
LIN {X 0,Y 319.932,Z 380.629,A -85,B 0,C 180,E1 -15306.663,E2 -15306.663} C_VEL
LIN {X 0,Y 319.76,Z 380.651,A -85,B 0,C 180,E1 -15310.127,E2 -15310.127} C_VEL
LIN {X 0,Y 319.731,Z 380.656,A -85,B 0,C 180,E1 -15314.724,E2 -15314.724} C_VEL
LIN {X 0,Y 319.689,Z 380.664,A -85,B 0,C 180,E1 -15319.038,E2 -15319.038} C_VEL
LIN {X 0,Y 319.571,Z 380.678,A -85,B 0,C 180,E1 -15323.319,E2 -15323.319} C_VEL
LIN {X 0,Y 319.635,Z 380.667,A -85,B 0,C 180,E1 -15326.088,E2 -15326.088} C_VEL
LIN {X 0,Y 319.59,Z 380.677,A -85,B 0,C 180,E1 -15328.934,E2 -15328.934} C_VEL
LIN {X 0,Y 319.534,Z 380.679,A -85,B 0,C 180,E1 -15331.862,E2 -15331.862} C_VEL
LIN {X 0,Y 319.581,Z 380.674,A -85,B 0,C 180,E1 -15335.543,E2 -15335.543} C_VEL
LIN {X 0,Y 319.558,Z 380.676,A -85,B 0,C 180,E1 -15338.01,E2 -15338.01} C_VEL
LIN {X 0,Y 319.527,Z 380.68,A -85,B 0,C 180,E1 -15341.597,E2 -15341.597} C_VEL
LIN {X 0,Y 319.516,Z 380.687,A -85,B 0,C 180,E1 -15344.738,E2 -15344.738} C_VEL
LIN {X 0,Y 319.527,Z 380.683,A -85,B 0,C 180,E1 -15348.403,E2 -15348.403} C_VEL
LIN {X 0,Y 319.579,Z 380.677,A -85,B 0,C 180,E1 -15352.344,E2 -15352.344} C_VEL
LIN {X 0,Y 319.561,Z 380.677,A -85,B 0,C 180,E1 -15355.124,E2 -15355.124} C_VEL
LIN {X 0,Y 319.567,Z 380.676,A -85,B 0,C 180,E1 -15359.059,E2 -15359.059} C_VEL
LIN {X 0,Y 319.607,Z 380.676,A -85,B 0,C 180,E1 -15362.498,E2 -15362.498} C_VEL
LIN {X 0,Y 319.607,Z 380.67,A -85,B 0,C 180,E1 -15365.304,E2 -15365.304} C_VEL
LIN {X 0,Y 319.624,Z 380.668,A -85,B 0,C 180,E1 -15369.402,E2 -15369.402} C_VEL
LIN {X 0,Y 319.661,Z 380.667,A -85,B 0,C 180,E1 -15372.073,E2 -15372.073} C_VEL
LIN {X 0,Y 319.734,Z 380.658,A -85,B 0,C 180,E1 -15376.008,E2 -15376.008} C_VEL
LIN {X 0,Y 319.76,Z 380.654,A -85,B 0,C 180,E1 -15379.873,E2 -15379.873} C_VEL
LIN {X 0,Y 319.927,Z 380.633,A -85,B 0,C 180,E1 -15382.426,E2 -15382.426} C_VEL
LIN {X 0,Y 319.748,Z 380.653,A -85,B 0,C 180,E1 -15384.956,E2 -15384.956} C_VEL
LIN {X 0,Y 319.993,Z 380.623,A -85,B 0,C 180,E1 -15387.483,E2 -15387.483} C_VEL
LIN {X 0,Y 320.171,Z 380.606,A -85,B 0,C 180,E1 -15390,E2 -15390} C_VEL
LIN {X 0,Y 319.992,Z 380.623,A -85,B 0,C 180,E1 -15392.518,E2 -15392.518} C_VEL
LIN {X 0,Y 319.946,Z 380.63,A -85,B 0,C 180,E1 -15396.306,E2 -15396.306} C_VEL
LIN {X 0,Y 319.84,Z 380.641,A -85,B 0,C 180,E1 -15398.848,E2 -15398.848} C_VEL
LIN {X 0,Y 319.684,Z 380.661,A -85,B 0,C 180,E1 -15402.7,E2 -15402.7} C_VEL
LIN {X 0,Y 319.702,Z 380.66,A -85,B 0,C 180,E1 -15405.296,E2 -15405.296} C_VEL
LIN {X 0,Y 319.677,Z 380.663,A -85,B 0,C 180,E1 -15409.255,E2 -15409.255} C_VEL
LIN {X 0,Y 319.573,Z 380.677,A -85,B 0,C 180,E1 -15413.32,E2 -15413.32} C_VEL
LIN {X 0,Y 319.637,Z 380.668,A -85,B 0,C 180,E1 -15416.088,E2 -15416.088} C_VEL
LIN {X 0,Y 319.582,Z 380.674,A -85,B 0,C 180,E1 -15418.935,E2 -15418.935} C_VEL
LIN {X 0,Y 319.533,Z 380.682,A -85,B 0,C 180,E1 -15421.862,E2 -15421.862} C_VEL
LIN {X 0,Y 319.583,Z 380.678,A -85,B 0,C 180,E1 -15425.543,E2 -15425.543} C_VEL
LIN {X 0,Y 319.576,Z 380.675,A -85,B 0,C 180,E1 -15428.008,E2 -15428.008} C_VEL
LIN {X 0,Y 319.528,Z 380.683,A -85,B 0,C 180,E1 -15431.597,E2 -15431.597} C_VEL
LIN {X 0,Y 319.518,Z 380.687,A -85,B 0,C 180,E1 -15435.262,E2 -15435.262} C_VEL
LIN {X 0,Y 319.531,Z 380.681,A -85,B 0,C 180,E1 -15438.712,E2 -15438.712} C_VEL
LIN {X 0,Y 319.564,Z 380.676,A -85,B 0,C 180,E1 -15442.348,E2 -15442.348} C_VEL
LIN {X 0,Y 319.572,Z 380.68,A -85,B 0,C 180,E1 -15445.125,E2 -15445.125} C_VEL
LIN {X 0,Y 319.787,Z 380.683,A -85,B 0,C 180,E1 -15448.291,E2 -15448.291} C_VEL
LIN {X 0,Y 319.836,Z 385.009,A -85,B 0,C 180,E1 -15451.091,E2 -15451.091} C_VEL
LIN {X 0,Y 319.459,Z 390.326,A -85,B 0,C 180,E1 -15454.421,E2 -15454.421} C_VEL
LIN {X 0,Y 319.065,Z 397.222,A -85,B 0,C 180,E1 -15458.688,E2 -15458.688} C_VEL
LIN {X 0,Y 318.803,Z 403.857,A -85,B 0,C 180,E1 -15462.686,E2 -15462.686} C_VEL
LIN {X 0,Y 318.549,Z 410.62,A -85,B 0,C 180,E1 -15466.662,E2 -15466.662} C_VEL
LIN {X 0,Y 318.495,Z 412.47,A -85,B 0,C 180,E1 -15467.738,E2 -15467.738} C_VEL
LIN {X 0,Y 319.606,Z 423.429,A -85,B 0,C 180,E1 -15468.523,E2 -15468.523} C_VEL
LIN {X 0,Y 319.339,Z 428.802,A -85,B 0,C 180,E1 -15468.975,E2 -15468.975} C_VEL
LIN {X 0,Y 317.889,Z 433.93,A -85,B 0,C 180,E1 -15469.45,E2 -15469.45} C_VEL
LIN {X 0,Y 313.403,Z 445.167,A -85,B 0,C 180,E1 -15470.739,E2 -15470.739} C_VEL
LIN {X 0,Y 312.486,Z 449.769,A -85,B 0,C 180,E1 -15471.41,E2 -15471.41} C_VEL
LIN {X 0,Y 312.176,Z 458.194,A -85,B 0,C 180,E1 -15472.887,E2 -15472.887} C_VEL
LIN {X 0,Y 311.887,Z 465.472,A -85,B 0,C 180,E1 -15474.504,E2 -15474.504} C_VEL
LIN {X 0,Y 311.521,Z 471.178,A -85,B 0,C 180,E1 -15476.119,E2 -15476.119} C_VEL
LIN {X 0,Y 311.376,Z 476.283,A -85,B 0,C 180,E1 -15478.06,E2 -15478.06} C_VEL
LIN {X 0,Y 311.418,Z 479.747,A -85,B 0,C 180,E1 -15480,E2 -15480} C_VEL
LIN {X 0,Y 311.587,Z 481.219,A -85,B 0,C 180,E1 -15481.292,E2 -15481.292} C_VEL
LIN {X 0,Y 311.81,Z 482.051,A -85,B 0,C 180,E1 -15482.584,E2 -15482.584} C_VEL
LIN {X 0,Y 312.172,Z 482.243,A -85,B 0,C 180,E1 -15483.873,E2 -15483.873} C_VEL
LIN {X 0,Y 312.773,Z 481.799,A -85,B 0,C 180,E1 -15485.157,E2 -15485.157} C_VEL
LIN {X 0,Y 313.469,Z 480.734,A -85,B 0,C 180,E1 -15486.436,E2 -15486.436} C_VEL
LIN {X 0,Y 314.802,Z 477.969,A -85,B 0,C 180,E1 -15488.344,E2 -15488.344} C_VEL
LIN {X 0,Y 316.281,Z 473.704,A -85,B 0,C 180,E1 -15490.24,E2 -15490.24} C_VEL
LIN {X 0,Y 318.142,Z 467.686,A -85,B 0,C 180,E1 -15492.114,E2 -15492.114} C_VEL
LIN {X 0,Y 319.894,Z 461.235,A -85,B 0,C 180,E1 -15493.661,E2 -15493.661} C_VEL
LIN {X 0,Y 321.922,Z 453.037,A -85,B 0,C 180,E1 -15495.187,E2 -15495.187} C_VEL
LIN {X 0,Y 322.484,Z 449.614,A -85,B 0,C 180,E1 -15495.751,E2 -15495.751} C_VEL
LIN {X 0,Y 321.824,Z 442.652,A -85,B 0,C 180,E1 -15497.005,E2 -15497.005} C_VEL
LIN {X 0,Y 319.794,Z 433.557,A -85,B 0,C 180,E1 -15498.605,E2 -15498.605} C_VEL
LIN {X 0,Y 316.876,Z 424.762,A -85,B 0,C 180,E1 -15500.132,E2 -15500.132} C_VEL
LIN {X 0,Y 315.095,Z 419.904,A -85,B 0,C 180,E1 -15500.994,E2 -15500.994} C_VEL
LIN {X 0,Y 316.137,Z 415.724,A -85,B 0,C 180,E1 -15504.985,E2 -15504.985} C_VEL
LIN {X 0,Y 317.019,Z 413.155,A -85,B 0,C 180,E1 -15507.746,E2 -15507.746} C_VEL
LIN {X 0,Y 317.848,Z 410.904,A -85,B 0,C 180,E1 -15510.568,E2 -15510.568} C_VEL
LIN {X 0,Y 318.352,Z 409.155,A -85,B 0,C 180,E1 -15513.498,E2 -15513.498} C_VEL
LIN {X 0,Y 318.574,Z 408.059,A -85,B 0,C 180,E1 -15516.559,E2 -15516.559} C_VEL
LIN {X 0,Y 318.775,Z 407.662,A -85,B 0,C 180,E1 -15519.744,E2 -15519.744} C_VEL
LIN {X 0,Y 319.153,Z 408.195,A -85,B 0,C 180,E1 -15523.39,E2 -15523.39} C_VEL
LIN {X 0,Y 319.629,Z 409.903,A -85,B 0,C 180,E1 -15527.029,E2 -15527.029} C_VEL
LIN {X 0,Y 319.978,Z 411.137,A -85,B 0,C 180,E1 -15528.782,E2 -15528.782} C_VEL
LIN {X 0,Y 320.629,Z 414.38,A -85,B 0,C 180,E1 -15532.139,E2 -15532.139} C_VEL
LIN {X 0,Y 321.624,Z 418.453,A -85,B 0,C 180,E1 -15535.379,E2 -15535.379} C_VEL
LIN {X 0,Y 322.036,Z 422.131,A -85,B 0,C 180,E1 -15537.678,E2 -15537.678} C_VEL
LIN {X 0,Y 321.852,Z 423.5,A -85,B 0,C 180,E1 -15538.394,E2 -15538.394} C_VEL
LIN {X 0,Y 319.16,Z 430.998,A -85,B 0,C 180,E1 -15541.741,E2 -15541.741} C_VEL
LIN {X 0,Y 317.485,Z 436.639,A -85,B 0,C 180,E1 -15544.052,E2 -15544.052} C_VEL
LIN {X 0,Y 320.418,Z 449.668,A -85,B 0,C 180,E1 -15545.371,E2 -15545.371} C_VEL
LIN {X 0,Y 321.868,Z 460.526,A -85,B 0,C 180,E1 -15546.502,E2 -15546.502} C_VEL
LIN {X 0,Y 322.078,Z 470.631,A -85,B 0,C 180,E1 -15547.592,E2 -15547.592} C_VEL
LIN {X 0,Y 320.896,Z 482.509,A -85,B 0,C 180,E1 -15548.984,E2 -15548.984} C_VEL
LIN {X 0,Y 318.618,Z 493.647,A -85,B 0,C 180,E1 -15550.511,E2 -15550.511} C_VEL
LIN {X 0,Y 316.49,Z 503.597,A -85,B 0,C 180,E1 -15552.221,E2 -15552.221} C_VEL
LIN {X 0,Y 314.596,Z 512.109,A -85,B 0,C 180,E1 -15554.053,E2 -15554.053} C_VEL
LIN {X 0,Y 313.174,Z 519.545,A -85,B 0,C 180,E1 -15556.04,E2 -15556.04} C_VEL
LIN {X 0,Y 311.862,Z 526.16,A -85,B 0,C 180,E1 -15558.298,E2 -15558.298} C_VEL
LIN {X 0,Y 311.31,Z 530.593,A -85,B 0,C 180,E1 -15560.252,E2 -15560.252} C_VEL
LIN {X 0,Y 311.09,Z 533.975,A -85,B 0,C 180,E1 -15562.209,E2 -15562.209} C_VEL
LIN {X 0,Y 311.078,Z 535.946,A -85,B 0,C 180,E1 -15563.757,E2 -15563.757} C_VEL
LIN {X 0,Y 311.128,Z 537.784,A -85,B 0,C 180,E1 -15566.114,E2 -15566.114} C_VEL
LIN {X 0,Y 311.335,Z 538.224,A -85,B 0,C 180,E1 -15567.412,E2 -15567.412} C_VEL
LIN {X 0,Y 311.504,Z 538.186,A -85,B 0,C 180,E1 -15568.707,E2 -15568.707} C_VEL
LIN {X 0,Y 311.485,Z 537.707,A -85,B 0,C 180,E1 -15570,E2 -15570} C_VEL
LIN {X 0,Y 311.538,Z 536.799,A -85,B 0,C 180,E1 -15571.292,E2 -15571.292} C_VEL
LIN {X 0,Y 311.616,Z 535.386,A -85,B 0,C 180,E1 -15572.585,E2 -15572.585} C_VEL
LIN {X 0,Y 311.446,Z 532.321,A -85,B 0,C 180,E1 -15574.53,E2 -15574.53} C_VEL
LIN {X 0,Y 311.421,Z 528.071,A -85,B 0,C 180,E1 -15576.479,E2 -15576.479} C_VEL
LIN {X 0,Y 311.506,Z 522.478,A -85,B 0,C 180,E1 -15578.433,E2 -15578.433} C_VEL
LIN {X 0,Y 311.701,Z 515.249,A -85,B 0,C 180,E1 -15580.392,E2 -15580.392} C_VEL
LIN {X 0,Y 312.107,Z 507.807,A -85,B 0,C 180,E1 -15582.022,E2 -15582.022} C_VEL
LIN {X 0,Y 312.689,Z 498.644,A -85,B 0,C 180,E1 -15583.65,E2 -15583.65} C_VEL
LIN {X 0,Y 313.491,Z 488.577,A -85,B 0,C 180,E1 -15585.088,E2 -15585.088} C_VEL
LIN {X 0,Y 314.156,Z 478.588,A -85,B 0,C 180,E1 -15586.238,E2 -15586.238} C_VEL
LIN {X 0,Y 314.395,Z 471.657,A -85,B 0,C 180,E1 -15586.894,E2 -15586.894} C_VEL
LIN {X 0,Y 313.579,Z 459.155,A -85,B 0,C 180,E1 -15587.864,E2 -15587.864} C_VEL
LIN {X 0,Y 312.795,Z 446.063,A -85,B 0,C 180,E1 -15588.586,E2 -15588.586} C_VEL
LIN {X 0,Y 312.571,Z 439.779,A -85,B 0,C 180,E1 -15588.852,E2 -15588.852} C_VEL
LIN {X 0,Y 314.297,Z 425.677,A -85,B 0,C 180,E1 -15593.734,E2 -15593.734} C_VEL
LIN {X 0,Y 316.507,Z 411.947,A -85,B 0,C 180,E1 -15598.516,E2 -15598.516} C_VEL
LIN {X 0,Y 317.471,Z 405.968,A -85,B 0,C 180,E1 -15600.608,E2 -15600.608} C_VEL
LIN {X 0,Y 315.807,Z 397.603,A -85,B 0,C 180,E1 -15603.804,E2 -15603.804} C_VEL
LIN {X 0,Y 313.801,Z 387.683,A -85,B 0,C 180,E1 -15607.739,E2 -15607.739} C_VEL
LIN {X 0,Y 312.53,Z 381.557,A -85,B 0,C 180,E1 -15610.363,E2 -15610.363} C_VEL
LIN {X 0,Y 312.512,Z 381.56,A -85,B 0,C 180,E1 -15614.199,E2 -15614.199} C_VEL
LIN {X 0,Y 312.488,Z 381.56,A -85,B 0,C 180,E1 -15617.918,E2 -15617.918} C_VEL
LIN {X 0,Y 312.536,Z 381.555,A -85,B 0,C 180,E1 -15621.91,E2 -15621.91} C_VEL
LIN {X 0,Y 312.507,Z 381.557,A -85,B 0,C 180,E1 -15625.79,E2 -15625.79} C_VEL
LIN {X 0,Y 312.521,Z 381.553,A -85,B 0,C 180,E1 -15628.854,E2 -15628.854} C_VEL
LIN {X 0,Y 312.57,Z 381.551,A -85,B 0,C 180,E1 -15631.824,E2 -15631.824} C_VEL
LIN {X 0,Y 312.586,Z 381.545,A -85,B 0,C 180,E1 -15634.711,E2 -15634.711} C_VEL
LIN {X 0,Y 312.588,Z 381.547,A -85,B 0,C 180,E1 -15637.529,E2 -15637.529} C_VEL
LIN {X 0,Y 312.639,Z 381.542,A -85,B 0,C 180,E1 -15641.656,E2 -15641.656} C_VEL
LIN {X 0,Y 312.694,Z 381.536,A -85,B 0,C 180,E1 -15645.686,E2 -15645.686} C_VEL
LIN {X 0,Y 312.703,Z 381.536,A -85,B 0,C 180,E1 -15649.642,E2 -15649.642} C_VEL
LIN {X 0,Y 312.873,Z 381.51,A -85,B 0,C 180,E1 -15652.254,E2 -15652.254} C_VEL
LIN {X 0,Y 312.72,Z 381.529,A -85,B 0,C 180,E1 -15654.842,E2 -15654.842} C_VEL
LIN {X 0,Y 312.953,Z 381.504,A -85,B 0,C 180,E1 -15657.426,E2 -15657.426} C_VEL
LIN {X 0,Y 313.104,Z 381.482,A -85,B 0,C 180,E1 -15660,E2 -15660} C_VEL
LIN {X 0,Y 312.937,Z 381.501,A -85,B 0,C 180,E1 -15662.574,E2 -15662.574} C_VEL
LIN {X 0,Y 312.895,Z 381.505,A -85,B 0,C 180,E1 -15666.646,E2 -15666.646} C_VEL
LIN {X 0,Y 312.789,Z 381.522,A -85,B 0,C 180,E1 -15669.049,E2 -15669.049} C_VEL
LIN {X 0,Y 312.638,Z 381.541,A -85,B 0,C 180,E1 -15672.991,E2 -15672.991} C_VEL
LIN {X 0,Y 312.639,Z 381.54,A -85,B 0,C 180,E1 -15675.65,E2 -15675.65} C_VEL
LIN {X 0,Y 312.631,Z 381.544,A -85,B 0,C 180,E1 -15679.237,E2 -15679.237} C_VEL
LIN {X 0,Y 312.546,Z 381.552,A -85,B 0,C 180,E1 -15682.789,E2 -15682.789} C_VEL
LIN {X 0,Y 312.603,Z 381.543,A -85,B 0,C 180,E1 -15685.936,E2 -15685.936} C_VEL
LIN {X 0,Y 312.546,Z 381.551,A -85,B 0,C 180,E1 -15689.65,E2 -15689.65} C_VEL
LIN {X 0,Y 312.52,Z 381.553,A -85,B 0,C 180,E1 -15693.689,E2 -15693.689} C_VEL
LIN {X 0,Y 312.526,Z 381.554,A -85,B 0,C 180,E1 -15697.385,E2 -15697.385} C_VEL
LIN {X 0,Y 312.49,Z 381.561,A -85,B 0,C 180,E1 -15700.709,E2 -15700.709} C_VEL
LIN {X 0,Y 312.474,Z 381.56,A -85,B 0,C 180,E1 -15704.206,E2 -15704.206} C_VEL
LIN {X 0,Y 312.486,Z 381.558,A -85,B 0,C 180,E1 -15707.918,E2 -15707.918} C_VEL
LIN {X 0,Y 312.536,Z 381.551,A -85,B 0,C 180,E1 -15711.911,E2 -15711.911} C_VEL
LIN {X 0,Y 312.507,Z 381.555,A -85,B 0,C 180,E1 -15715.79,E2 -15715.79} C_VEL
LIN {X 0,Y 312.521,Z 381.555,A -85,B 0,C 180,E1 -15718.854,E2 -15718.854} C_VEL
LIN {X 0,Y 312.571,Z 381.547,A -85,B 0,C 180,E1 -15721.825,E2 -15721.825} C_VEL
LIN {X 0,Y 312.587,Z 381.548,A -85,B 0,C 180,E1 -15724.711,E2 -15724.711} C_VEL
LIN {X 0,Y 312.589,Z 381.544,A -85,B 0,C 180,E1 -15727.529,E2 -15727.529} C_VEL
LIN {X 0,Y 312.641,Z 381.539,A -85,B 0,C 180,E1 -15731.657,E2 -15731.657} C_VEL
LIN {X 0,Y 312.696,Z 381.532,A -85,B 0,C 180,E1 -15735.687,E2 -15735.687} C_VEL
LIN {X 0,Y 312.704,Z 381.531,A -85,B 0,C 180,E1 -15739.642,E2 -15739.642} C_VEL
LIN {X 0,Y 312.868,Z 381.514,A -85,B 0,C 180,E1 -15742.254,E2 -15742.254} C_VEL
LIN {X 0,Y 312.718,Z 381.529,A -85,B 0,C 180,E1 -15744.843,E2 -15744.843} C_VEL
LIN {X 0,Y 312.993,Z 381.495,A -85,B 0,C 180,E1 -15748.714,E2 -15748.714} C_VEL
LIN {X 0,Y 313.123,Z 381.484,A -85,B 0,C 180,E1 -15750,E2 -15750} C_VEL
LIN {X 0,Y 312.939,Z 381.502,A -85,B 0,C 180,E1 -15752.575,E2 -15752.575} C_VEL
LIN {X 0,Y 312.903,Z 381.506,A -85,B 0,C 180,E1 -15756.448,E2 -15756.448} C_VEL
LIN {X 0,Y 312.769,Z 381.522,A -85,B 0,C 180,E1 -15759.05,E2 -15759.05} C_VEL
LIN {X 0,Y 312.637,Z 381.538,A -85,B 0,C 180,E1 -15762.991,E2 -15762.991} C_VEL
LIN {X 0,Y 312.641,Z 381.543,A -85,B 0,C 180,E1 -15765.65,E2 -15765.65} C_VEL
LIN {X 0,Y 312.633,Z 381.541,A -85,B 0,C 180,E1 -15769.237,E2 -15769.237} C_VEL
LIN {X 0,Y 312.549,Z 381.55,A -85,B 0,C 180,E1 -15772.789,E2 -15772.789} C_VEL
LIN {X 0,Y 312.605,Z 381.545,A -85,B 0,C 180,E1 -15775.936,E2 -15775.936} C_VEL
LIN {X 0,Y 312.54,Z 381.554,A -85,B 0,C 180,E1 -15779.651,E2 -15779.651} C_VEL
LIN {X 0,Y 312.522,Z 381.556,A -85,B 0,C 180,E1 -15783.689,E2 -15783.689} C_VEL
LIN {X 0,Y 312.54,Z 381.556,A -85,B 0,C 180,E1 -15787.383,E2 -15787.383} C_VEL
LIN {X 0,Y 312.493,Z 381.557,A -85,B 0,C 180,E1 -15790.709,E2 -15790.709} C_VEL
LIN {X 0,Y 312.475,Z 381.559,A -85,B 0,C 180,E1 -15794.206,E2 -15794.206} C_VEL
LIN {X 0,Y 312.488,Z 381.557,A -85,B 0,C 180,E1 -15797.918,E2 -15797.918} C_VEL
LIN {X 0,Y 312.508,Z 381.555,A -85,B 0,C 180,E1 -15801.917,E2 -15801.917} C_VEL
LIN {X 0,Y 312.531,Z 381.552,A -85,B 0,C 180,E1 -15805.793,E2 -15805.793} C_VEL
LIN {X 0,Y 312.71,Z 381.556,A -85,B 0,C 180,E1 -15808.213,E2 -15808.213} C_VEL
LIN {X 0,Y 312.879,Z 384.808,A -85,B 0,C 180,E1 -15810.385,E2 -15810.385} C_VEL
LIN {X 0,Y 312.426,Z 390.66,A -85,B 0,C 180,E1 -15814.132,E2 -15814.132} C_VEL
LIN {X 0,Y 312.022,Z 397.136,A -85,B 0,C 180,E1 -15818.183,E2 -15818.183} C_VEL
LIN {X 0,Y 311.78,Z 402.685,A -85,B 0,C 180,E1 -15821.604,E2 -15821.604} C_VEL
LIN {X 0,Y 311.533,Z 409.906,A -85,B 0,C 180,E1 -15825.944,E2 -15825.944} C_VEL
LIN {X 0,Y 311.43,Z 412.743,A -85,B 0,C 180,E1 -15827.62,E2 -15827.62} C_VEL
LIN {X 0,Y 312.61,Z 424.598,A -85,B 0,C 180,E1 -15828.491,E2 -15828.491} C_VEL
LIN {X 0,Y 313.345,Z 431.934,A -85,B 0,C 180,E1 -15829.173,E2 -15829.173} C_VEL
LIN {X 0,Y 312.834,Z 441.904,A -85,B 0,C 180,E1 -15830.3,E2 -15830.3} C_VEL
LIN {X 0,Y 312.486,Z 449.769,A -85,B 0,C 180,E1 -15831.41,E2 -15831.41} C_VEL
LIN {X 0,Y 311.617,Z 454.151,A -85,B 0,C 180,E1 -15832.122,E2 -15832.122} C_VEL
LIN {X 0,Y 308.504,Z 460.745,A -85,B 0,C 180,E1 -15833.366,E2 -15833.366} C_VEL
LIN {X 0,Y 305.402,Z 466.685,A -85,B 0,C 180,E1 -15834.747,E2 -15834.747} C_VEL
LIN {X 0,Y 304.564,Z 469.966,A -85,B 0,C 180,E1 -15835.66,E2 -15835.66} C_VEL
LIN {X 0,Y 304.299,Z 474.892,A -85,B 0,C 180,E1 -15837.352,E2 -15837.352} C_VEL
LIN {X 0,Y 304.292,Z 479.088,A -85,B 0,C 180,E1 -15839.338,E2 -15839.338} C_VEL
LIN {X 0,Y 304.514,Z 481.75,A -85,B 0,C 180,E1 -15841.322,E2 -15841.322} C_VEL
LIN {X 0,Y 304.776,Z 482.727,A -85,B 0,C 180,E1 -15842.643,E2 -15842.643} C_VEL
LIN {X 0,Y 305.149,Z 483.077,A -85,B 0,C 180,E1 -15843.962,E2 -15843.962} C_VEL
LIN {X 0,Y 305.773,Z 482.802,A -85,B 0,C 180,E1 -15845.275,E2 -15845.275} C_VEL
LIN {X 0,Y 306.511,Z 481.905,A -85,B 0,C 180,E1 -15846.583,E2 -15846.583} C_VEL
LIN {X 0,Y 307.901,Z 479.362,A -85,B 0,C 180,E1 -15848.532,E2 -15848.532} C_VEL
LIN {X 0,Y 309.479,Z 475.352,A -85,B 0,C 180,E1 -15850.467,E2 -15850.467} C_VEL
LIN {X 0,Y 311.449,Z 469.75,A -85,B 0,C 180,E1 -15852.379,E2 -15852.379} C_VEL
LIN {X 0,Y 313.28,Z 463.631,A -85,B 0,C 180,E1 -15853.955,E2 -15853.955} C_VEL
LIN {X 0,Y 315.398,Z 455.862,A -85,B 0,C 180,E1 -15855.509,E2 -15855.509} C_VEL
LIN {X 0,Y 316.266,Z 451.578,A -85,B 0,C 180,E1 -15856.271,E2 -15856.271} C_VEL
LIN {X 0,Y 315.771,Z 445.328,A -85,B 0,C 180,E1 -15857.485,E2 -15857.485} C_VEL
LIN {X 0,Y 313.989,Z 436.617,A -85,B 0,C 180,E1 -15859.133,E2 -15859.133} C_VEL
LIN {X 0,Y 311.211,Z 427.72,A -85,B 0,C 180,E1 -15860.801,E2 -15860.801} C_VEL
LIN {X 0,Y 308.531,Z 420.596,A -85,B 0,C 180,E1 -15862.2,E2 -15862.2} C_VEL
LIN {X 0,Y 309.496,Z 417.264,A -85,B 0,C 180,E1 -15865.56,E2 -15865.56} C_VEL
LIN {X 0,Y 310.406,Z 414.8,A -85,B 0,C 180,E1 -15868.39,E2 -15868.39} C_VEL
LIN {X 0,Y 311.249,Z 412.734,A -85,B 0,C 180,E1 -15871.288,E2 -15871.288} C_VEL
LIN {X 0,Y 311.674,Z 411.545,A -85,B 0,C 180,E1 -15873.454,E2 -15873.454} C_VEL
LIN {X 0,Y 311.869,Z 410.693,A -85,B 0,C 180,E1 -15875.868,E2 -15875.868} C_VEL
LIN {X 0,Y 312.062,Z 410.187,A -85,B 0,C 180,E1 -15879.094,E2 -15879.094} C_VEL
LIN {X 0,Y 312.39,Z 410.505,A -85,B 0,C 180,E1 -15882.448,E2 -15882.448} C_VEL
LIN {X 0,Y 312.614,Z 411.031,A -85,B 0,C 180,E1 -15884.181,E2 -15884.181} C_VEL
LIN {X 0,Y 313.133,Z 412.983,A -85,B 0,C 180,E1 -15887.788,E2 -15887.788} C_VEL
LIN {X 0,Y 313.745,Z 415.891,A -85,B 0,C 180,E1 -15891.155,E2 -15891.155} C_VEL
LIN {X 0,Y 314.647,Z 419.739,A -85,B 0,C 180,E1 -15894.497,E2 -15894.497} C_VEL
LIN {X 0,Y 315.279,Z 423.208,A -85,B 0,C 180,E1 -15896.897,E2 -15896.897} C_VEL
LIN {X 0,Y 315.191,Z 424.958,A -85,B 0,C 180,E1 -15897.92,E2 -15897.92} C_VEL
LIN {X 0,Y 313.818,Z 428.751,A -85,B 0,C 180,E1 -15899.742,E2 -15899.742} C_VEL
LIN {X 0,Y 311.296,Z 436.35,A -85,B 0,C 180,E1 -15902.999,E2 -15902.999} C_VEL
LIN {X 0,Y 314.036,Z 448.058,A -85,B 0,C 180,E1 -15904.303,E2 -15904.303} C_VEL
LIN {X 0,Y 315.758,Z 460.996,A -85,B 0,C 180,E1 -15905.75,E2 -15905.75} C_VEL
LIN {X 0,Y 315.922,Z 470.718,A -85,B 0,C 180,E1 -15906.869,E2 -15906.869} C_VEL
LIN {X 0,Y 314.822,Z 481.677,A -85,B 0,C 180,E1 -15908.214,E2 -15908.214} C_VEL
LIN {X 0,Y 312.711,Z 491.75,A -85,B 0,C 180,E1 -15909.613,E2 -15909.613} C_VEL
LIN {X 0,Y 310.561,Z 500.979,A -85,B 0,C 180,E1 -15911.187,E2 -15911.187} C_VEL
LIN {X 0,Y 308.359,Z 509.977,A -85,B 0,C 180,E1 -15913.079,E2 -15913.079} C_VEL
LIN {X 0,Y 306.718,Z 517.467,A -85,B 0,C 180,E1 -15915.061,E2 -15915.061} C_VEL
LIN {X 0,Y 305.267,Z 524.372,A -85,B 0,C 180,E1 -15917.366,E2 -15917.366} C_VEL
LIN {X 0,Y 304.443,Z 528.992,A -85,B 0,C 180,E1 -15919.357,E2 -15919.357} C_VEL
LIN {X 0,Y 304.017,Z 533.547,A -85,B 0,C 180,E1 -15922.027,E2 -15922.027} C_VEL
LIN {X 0,Y 304.01,Z 535.535,A -85,B 0,C 180,E1 -15923.752,E2 -15923.752} C_VEL
LIN {X 0,Y 304.046,Z 537.105,A -85,B 0,C 180,E1 -15926.023,E2 -15926.023} C_VEL
LIN {X 0,Y 304.267,Z 537.431,A -85,B 0,C 180,E1 -15927.352,E2 -15927.352} C_VEL
LIN {X 0,Y 304.457,Z 537.336,A -85,B 0,C 180,E1 -15928.677,E2 -15928.677} C_VEL
LIN {X 0,Y 304.444,Z 536.796,A -85,B 0,C 180,E1 -15930,E2 -15930} C_VEL
LIN {X 0,Y 304.507,Z 535.766,A -85,B 0,C 180,E1 -15931.322,E2 -15931.322} C_VEL
LIN {X 0,Y 304.491,Z 533.342,A -85,B 0,C 180,E1 -15933.308,E2 -15933.308} C_VEL
LIN {X 0,Y 304.405,Z 529.751,A -85,B 0,C 180,E1 -15935.299,E2 -15935.299} C_VEL
LIN {X 0,Y 304.439,Z 525.093,A -85,B 0,C 180,E1 -15937.228,E2 -15937.228} C_VEL
LIN {X 0,Y 304.528,Z 518.591,A -85,B 0,C 180,E1 -15939.297,E2 -15939.297} C_VEL
LIN {X 0,Y 304.869,Z 510.548,A -85,B 0,C 180,E1 -15941.3,E2 -15941.3} C_VEL
LIN {X 0,Y 305.393,Z 502.193,A -85,B 0,C 180,E1 -15942.966,E2 -15942.966} C_VEL
LIN {X 0,Y 306.048,Z 491.761,A -85,B 0,C 180,E1 -15944.631,E2 -15944.631} C_VEL
LIN {X 0,Y 306.874,Z 481.385,A -85,B 0,C 180,E1 -15945.951,E2 -15945.951} C_VEL
LIN {X 0,Y 307.382,Z 473.451,A -85,B 0,C 180,E1 -15946.777,E2 -15946.777} C_VEL
LIN {X 0,Y 306.64,Z 461.669,A -85,B 0,C 180,E1 -15947.765,E2 -15947.765} C_VEL
LIN {X 0,Y 305.816,Z 449.154,A -85,B 0,C 180,E1 -15948.551,E2 -15948.551} C_VEL
LIN {X 0,Y 305.508,Z 439.576,A -85,B 0,C 180,E1 -15948.984,E2 -15948.984} C_VEL
LIN {X 0,Y 307.43,Z 424.657,A -85,B 0,C 180,E1 -15954.298,E2 -15954.298} C_VEL
LIN {X 0,Y 309.762,Z 411.002,A -85,B 0,C 180,E1 -15959.196,E2 -15959.196} C_VEL
LIN {X 0,Y 310.456,Z 406.956,A -85,B 0,C 180,E1 -15960.657,E2 -15960.657} C_VEL
LIN {X 0,Y 308.576,Z 397.568,A -85,B 0,C 180,E1 -15964.312,E2 -15964.312} C_VEL
LIN {X 0,Y 306.649,Z 388.023,A -85,B 0,C 180,E1 -15968.229,E2 -15968.229} C_VEL
LIN {X 0,Y 305.501,Z 382.432,A -85,B 0,C 180,E1 -15970.662,E2 -15970.662} C_VEL
LIN {X 0,Y 305.448,Z 382.437,A -85,B 0,C 180,E1 -15974.498,E2 -15974.498} C_VEL
LIN {X 0,Y 305.444,Z 382.439,A -85,B 0,C 180,E1 -15978.144,E2 -15978.144} C_VEL
LIN {X 0,Y 305.496,Z 382.429,A -85,B 0,C 180,E1 -15981.6,E2 -15981.6} C_VEL
LIN {X 0,Y 305.463,Z 382.432,A -85,B 0,C 180,E1 -15984.887,E2 -15984.887} C_VEL
LIN {X 0,Y 305.45,Z 382.436,A -85,B 0,C 180,E1 -15988.355,E2 -15988.355} C_VEL
LIN {X 0,Y 305.513,Z 382.426,A -85,B 0,C 180,E1 -15991.113,E2 -15991.113} C_VEL
LIN {X 0,Y 305.571,Z 382.422,A -85,B 0,C 180,E1 -15994.088,E2 -15994.088} C_VEL
LIN {X 0,Y 305.501,Z 382.429,A -85,B 0,C 180,E1 -15998.403,E2 -15998.403} C_VEL
LIN {X 0,Y 305.591,Z 382.417,A -85,B 0,C 180,E1 -16001.218,E2 -16001.218} C_VEL
LIN {X 0,Y 305.649,Z 382.411,A -85,B 0,C 180,E1 -16005.349,E2 -16005.349} C_VEL
LIN {X 0,Y 305.639,Z 382.413,A -85,B 0,C 180,E1 -16009.4,E2 -16009.4} C_VEL
LIN {X 0,Y 305.814,Z 382.39,A -85,B 0,C 180,E1 -16012.074,E2 -16012.074} C_VEL
LIN {X 0,Y 305.691,Z 382.404,A -85,B 0,C 180,E1 -16014.724,E2 -16014.724} C_VEL
LIN {X 0,Y 305.96,Z 382.37,A -85,B 0,C 180,E1 -16018.684,E2 -16018.684} C_VEL
LIN {X 0,Y 305.958,Z 382.374,A -85,B 0,C 180,E1 -16021.316,E2 -16021.316} C_VEL
LIN {X 0,Y 305.851,Z 382.384,A -85,B 0,C 180,E1 -16026.625,E2 -16026.625} C_VEL
LIN {X 0,Y 305.737,Z 382.402,A -85,B 0,C 180,E1 -16029.26,E2 -16029.26} C_VEL
LIN {X 0,Y 305.592,Z 382.421,A -85,B 0,C 180,E1 -16033.296,E2 -16033.296} C_VEL
LIN {X 0,Y 305.595,Z 382.416,A -85,B 0,C 180,E1 -16036.02,E2 -16036.02} C_VEL
LIN {X 0,Y 305.577,Z 382.421,A -85,B 0,C 180,E1 -16039.445,E2 -16039.445} C_VEL
LIN {X 0,Y 305.492,Z 382.434,A -85,B 0,C 180,E1 -16043.042,E2 -16043.042} C_VEL
LIN {X 0,Y 305.548,Z 382.421,A -85,B 0,C 180,E1 -16046.227,E2 -16046.227} C_VEL
LIN {X 0,Y 305.497,Z 382.433,A -85,B 0,C 180,E1 -16049.05,E2 -16049.05} C_VEL
LIN {X 0,Y 305.445,Z 382.434,A -85,B 0,C 180,E1 -16051.952,E2 -16051.952} C_VEL
LIN {X 0,Y 305.463,Z 382.436,A -85,B 0,C 180,E1 -16055.113,E2 -16055.113} C_VEL
LIN {X 0,Y 305.45,Z 382.436,A -85,B 0,C 180,E1 -16058.529,E2 -16058.529} C_VEL
LIN {X 0,Y 305.46,Z 382.436,A -85,B 0,C 180,E1 -16062.587,E2 -16062.587} C_VEL
LIN {X 0,Y 305.443,Z 382.437,A -85,B 0,C 180,E1 -16066.348,E2 -16066.348} C_VEL
LIN {X 0,Y 305.459,Z 382.433,A -85,B 0,C 180,E1 -16069.893,E2 -16069.893} C_VEL
LIN {X 0,Y 305.5,Z 382.427,A -85,B 0,C 180,E1 -16073.627,E2 -16073.627} C_VEL
LIN {X 0,Y 305.466,Z 382.437,A -85,B 0,C 180,E1 -16076.484,E2 -16076.484} C_VEL
LIN {X 0,Y 305.459,Z 382.432,A -85,B 0,C 180,E1 -16079.591,E2 -16079.591} C_VEL
LIN {X 0,Y 305.52,Z 382.429,A -85,B 0,C 180,E1 -16082.609,E2 -16082.609} C_VEL
LIN {X 0,Y 305.51,Z 382.426,A -85,B 0,C 180,E1 -16085.539,E2 -16085.539} C_VEL
LIN {X 0,Y 305.532,Z 382.425,A -85,B 0,C 180,E1 -16089.816,E2 -16089.816} C_VEL
LIN {X 0,Y 305.578,Z 382.421,A -85,B 0,C 180,E1 -16092.603,E2 -16092.603} C_VEL
LIN {X 0,Y 305.651,Z 382.409,A -85,B 0,C 180,E1 -16095.349,E2 -16095.349} C_VEL
LIN {X 0,Y 305.641,Z 382.41,A -85,B 0,C 180,E1 -16099.4,E2 -16099.4} C_VEL
LIN {X 0,Y 305.811,Z 382.394,A -85,B 0,C 180,E1 -16102.075,E2 -16102.075} C_VEL
LIN {X 0,Y 305.689,Z 382.404,A -85,B 0,C 180,E1 -16104.724,E2 -16104.724} C_VEL
LIN {X 0,Y 305.96,Z 382.371,A -85,B 0,C 180,E1 -16108.684,E2 -16108.684} C_VEL
LIN {X 0,Y 305.96,Z 382.371,A -85,B 0,C 180,E1 -16111.316,E2 -16111.316} C_VEL
LIN {X 0,Y 305.845,Z 382.385,A -85,B 0,C 180,E1 -16116.598,E2 -16116.598} C_VEL
LIN {X 0,Y 305.706,Z 382.403,A -85,B 0,C 180,E1 -16119.261,E2 -16119.261} C_VEL
LIN {X 0,Y 305.592,Z 382.417,A -85,B 0,C 180,E1 -16123.296,E2 -16123.296} C_VEL
LIN {X 0,Y 305.597,Z 382.418,A -85,B 0,C 180,E1 -16126.02,E2 -16126.02} C_VEL
LIN {X 0,Y 305.58,Z 382.421,A -85,B 0,C 180,E1 -16129.445,E2 -16129.445} C_VEL
LIN {X 0,Y 305.493,Z 382.429,A -85,B 0,C 180,E1 -16133.042,E2 -16133.042} C_VEL
LIN {X 0,Y 305.534,Z 382.424,A -85,B 0,C 180,E1 -16136.221,E2 -16136.221} C_VEL
LIN {X 0,Y 305.49,Z 382.43,A -85,B 0,C 180,E1 -16139.048,E2 -16139.048} C_VEL
LIN {X 0,Y 305.444,Z 382.436,A -85,B 0,C 180,E1 -16141.952,E2 -16141.952} C_VEL
LIN {X 0,Y 305.465,Z 382.435,A -85,B 0,C 180,E1 -16145.113,E2 -16145.113} C_VEL
LIN {X 0,Y 305.47,Z 382.431,A -85,B 0,C 180,E1 -16148.533,E2 -16148.533} C_VEL
LIN {X 0,Y 305.461,Z 382.433,A -85,B 0,C 180,E1 -16152.587,E2 -16152.587} C_VEL
LIN {X 0,Y 305.445,Z 382.434,A -85,B 0,C 180,E1 -16156.348,E2 -16156.348} C_VEL
LIN {X 0,Y 305.46,Z 382.433,A -85,B 0,C 180,E1 -16159.893,E2 -16159.893} C_VEL
LIN {X 0,Y 305.485,Z 382.43,A -85,B 0,C 180,E1 -16163.631,E2 -16163.631} C_VEL
LIN {X 0,Y 305.702,Z 382.605,A -85,B 0,C 180,E1 -16168.28,E2 -16168.28} C_VEL
LIN {X 0,Y 305.769,Z 386.496,A -85,B 0,C 180,E1 -16170.859,E2 -16170.859} C_VEL
LIN {X 0,Y 305.305,Z 392.547,A -85,B 0,C 180,E1 -16174.795,E2 -16174.795} C_VEL
LIN {X 0,Y 304.907,Z 399.276,A -85,B 0,C 180,E1 -16179.067,E2 -16179.067} C_VEL
LIN {X 0,Y 304.647,Z 404.877,A -85,B 0,C 180,E1 -16182.548,E2 -16182.548} C_VEL
LIN {X 0,Y 304.377,Z 411.649,A -85,B 0,C 180,E1 -16186.65,E2 -16186.65} C_VEL
LIN {X 0,Y 304.354,Z 413.132,A -85,B 0,C 180,E1 -16187.54,E2 -16187.54} C_VEL
LIN {X 0,Y 305.489,Z 424.618,A -85,B 0,C 180,E1 -16188.387,E2 -16188.387} C_VEL
LIN {X 0,Y 306.258,Z 432.024,A -85,B 0,C 180,E1 -16189.087,E2 -16189.087} C_VEL
LIN {X 0,Y 305.755,Z 442.072,A -85,B 0,C 180,E1 -16190.24,E2 -16190.24} C_VEL
LIN {X 0,Y 305.363,Z 451.179,A -85,B 0,C 180,E1 -16191.564,E2 -16191.564} C_VEL
LIN {X 0,Y 305.07,Z 459.466,A -85,B 0,C 180,E1 -16193.077,E2 -16193.077} C_VEL
LIN {X 0,Y 304.749,Z 466.544,A -85,B 0,C 180,E1 -16194.707,E2 -16194.707} C_VEL
LIN {X 0,Y 304.564,Z 469.966,A -85,B 0,C 180,E1 -16195.66,E2 -16195.66} C_VEL
LIN {X 0,Y 303.732,Z 472.967,A -85,B 0,C 180,E1 -16196.606,E2 -16196.606} C_VEL
LIN {X 0,Y 300.735,Z 477.076,A -85,B 0,C 180,E1 -16198.219,E2 -16198.219} C_VEL
LIN {X 0,Y 297.921,Z 480.386,A -85,B 0,C 180,E1 -16199.939,E2 -16199.939} C_VEL
LIN {X 0,Y 297.39,Z 481.851,A -85,B 0,C 180,E1 -16201.035,E2 -16201.035} C_VEL
LIN {X 0,Y 297.743,Z 483.396,A -85,B 0,C 180,E1 -16202.706,E2 -16202.706} C_VEL
LIN {X 0,Y 298.128,Z 483.898,A -85,B 0,C 180,E1 -16204.055,E2 -16204.055} C_VEL
LIN {X 0,Y 298.769,Z 483.758,A -85,B 0,C 180,E1 -16205.399,E2 -16205.399} C_VEL
LIN {X 0,Y 299.544,Z 483.01,A -85,B 0,C 180,E1 -16206.737,E2 -16206.737} C_VEL
LIN {X 0,Y 300.451,Z 481.651,A -85,B 0,C 180,E1 -16208.068,E2 -16208.068} C_VEL
LIN {X 0,Y 302.131,Z 478.453,A -85,B 0,C 180,E1 -16210.047,E2 -16210.047} C_VEL
LIN {X 0,Y 304.015,Z 473.737,A -85,B 0,C 180,E1 -16212.008,E2 -16212.008} C_VEL
LIN {X 0,Y 306.246,Z 467.27,A -85,B 0,C 180,E1 -16213.943,E2 -16213.943} C_VEL
LIN {X 0,Y 308.412,Z 460.391,A -85,B 0,C 180,E1 -16215.531,E2 -16215.531} C_VEL
LIN {X 0,Y 309.997,Z 454.651,A -85,B 0,C 180,E1 -16216.61,E2 -16216.61} C_VEL
LIN {X 0,Y 309.873,Z 449.248,A -85,B 0,C 180,E1 -16217.716,E2 -16217.716} C_VEL
LIN {X 0,Y 308.621,Z 441.258,A -85,B 0,C 180,E1 -16219.361,E2 -16219.361} C_VEL
LIN {X 0,Y 305.888,Z 431.434,A -85,B 0,C 180,E1 -16221.362,E2 -16221.362} C_VEL
LIN {X 0,Y 303.104,Z 424.415,A -85,B 0,C 180,E1 -16222.854,E2 -16222.854} C_VEL
LIN {X 0,Y 302.025,Z 421.377,A -85,B 0,C 180,E1 -16223.484,E2 -16223.484} C_VEL
LIN {X 0,Y 303.37,Z 417.661,A -85,B 0,C 180,E1 -16227.602,E2 -16227.602} C_VEL
LIN {X 0,Y 304.556,Z 415.02,A -85,B 0,C 180,E1 -16231.37,E2 -16231.37} C_VEL
LIN {X 0,Y 305.017,Z 413.743,A -85,B 0,C 180,E1 -16233.953,E2 -16233.953} C_VEL
LIN {X 0,Y 305.246,Z 412.932,A -85,B 0,C 180,E1 -16236.772,E2 -16236.772} C_VEL
LIN {X 0,Y 305.561,Z 412.732,A -85,B 0,C 180,E1 -16240.092,E2 -16240.092} C_VEL
LIN {X 0,Y 305.923,Z 413.424,A -85,B 0,C 180,E1 -16243.566,E2 -16243.566} C_VEL
LIN {X 0,Y 306.418,Z 415.214,A -85,B 0,C 180,E1 -16247.219,E2 -16247.219} C_VEL
LIN {X 0,Y 306.907,Z 417.431,A -85,B 0,C 180,E1 -16250.119,E2 -16250.119} C_VEL
LIN {X 0,Y 307.752,Z 421.065,A -85,B 0,C 180,E1 -16253.576,E2 -16253.576} C_VEL
LIN {X 0,Y 308.464,Z 424.32,A -85,B 0,C 180,E1 -16256.068,E2 -16256.068} C_VEL
LIN {X 0,Y 308.565,Z 426.478,A -85,B 0,C 180,E1 -16257.43,E2 -16257.43} C_VEL
LIN {X 0,Y 308.1,Z 428.196,A -85,B 0,C 180,E1 -16258.355,E2 -16258.355} C_VEL
LIN {X 0,Y 305.23,Z 435.725,A -85,B 0,C 180,E1 -16261.811,E2 -16261.811} C_VEL
LIN {X 0,Y 308.481,Z 450.558,A -85,B 0,C 180,E1 -16263.623,E2 -16263.623} C_VEL
LIN {X 0,Y 309.845,Z 463.03,A -85,B 0,C 180,E1 -16265.134,E2 -16265.134} C_VEL
LIN {X 0,Y 309.749,Z 473.054,A -85,B 0,C 180,E1 -16266.372,E2 -16266.372} C_VEL
LIN {X 0,Y 308.426,Z 483.381,A -85,B 0,C 180,E1 -16267.739,E2 -16267.739} C_VEL
LIN {X 0,Y 306.147,Z 492.962,A -85,B 0,C 180,E1 -16269.156,E2 -16269.156} C_VEL
LIN {X 0,Y 304.321,Z 500.156,A -85,B 0,C 180,E1 -16270.435,E2 -16270.435} C_VEL
LIN {X 0,Y 301.916,Z 509.218,A -85,B 0,C 180,E1 -16272.385,E2 -16272.385} C_VEL
LIN {X 0,Y 300.031,Z 516.575,A -85,B 0,C 180,E1 -16274.372,E2 -16274.372} C_VEL
LIN {X 0,Y 298.732,Z 522.577,A -85,B 0,C 180,E1 -16276.393,E2 -16276.393} C_VEL
LIN {X 0,Y 297.615,Z 527.401,A -85,B 0,C 180,E1 -16278.42,E2 -16278.42} C_VEL
LIN {X 0,Y 297.09,Z 531.149,A -85,B 0,C 180,E1 -16280.468,E2 -16280.468} C_VEL
LIN {X 0,Y 296.92,Z 534.597,A -85,B 0,C 180,E1 -16283.203,E2 -16283.203} C_VEL
LIN {X 0,Y 296.935,Z 535.716,A -85,B 0,C 180,E1 -16284.567,E2 -16284.567} C_VEL
LIN {X 0,Y 297.2,Z 536.63,A -85,B 0,C 180,E1 -16287.289,E2 -16287.289} C_VEL
LIN {X 0,Y 297.41,Z 536.476,A -85,B 0,C 180,E1 -16288.646,E2 -16288.646} C_VEL
LIN {X 0,Y 297.412,Z 535.813,A -85,B 0,C 180,E1 -16290,E2 -16290} C_VEL
LIN {X 0,Y 297.477,Z 534.716,A -85,B 0,C 180,E1 -16291.354,E2 -16291.354} C_VEL
LIN {X 0,Y 297.46,Z 532.159,A -85,B 0,C 180,E1 -16293.386,E2 -16293.386} C_VEL
LIN {X 0,Y 297.373,Z 528.426,A -85,B 0,C 180,E1 -16295.424,E2 -16295.424} C_VEL
LIN {X 0,Y 297.393,Z 523.378,A -85,B 0,C 180,E1 -16297.467,E2 -16297.467} C_VEL
LIN {X 0,Y 297.485,Z 516.814,A -85,B 0,C 180,E1 -16299.519,E2 -16299.519} C_VEL
LIN {X 0,Y 297.818,Z 510.032,A -85,B 0,C 180,E1 -16301.226,E2 -16301.226} C_VEL
LIN {X 0,Y 298.327,Z 501.73,A -85,B 0,C 180,E1 -16302.932,E2 -16302.932} C_VEL
LIN {X 0,Y 298.974,Z 491.353,A -85,B 0,C 180,E1 -16304.637,E2 -16304.637} C_VEL
LIN {X 0,Y 299.825,Z 480.588,A -85,B 0,C 180,E1 -16306.042,E2 -16306.042} C_VEL
LIN {X 0,Y 300.266,Z 473.165,A -85,B 0,C 180,E1 -16306.837,E2 -16306.837} C_VEL
LIN {X 0,Y 299.535,Z 461.482,A -85,B 0,C 180,E1 -16307.847,E2 -16307.847} C_VEL
LIN {X 0,Y 298.728,Z 448.291,A -85,B 0,C 180,E1 -16308.696,E2 -16308.696} C_VEL
LIN {X 0,Y 298.442,Z 439.262,A -85,B 0,C 180,E1 -16309.116,E2 -16309.116} C_VEL
LIN {X 0,Y 300.379,Z 424.855,A -85,B 0,C 180,E1 -16314.418,E2 -16314.418} C_VEL
LIN {X 0,Y 302.633,Z 411.912,A -85,B 0,C 180,E1 -16319.188,E2 -16319.188} C_VEL
LIN {X 0,Y 303.37,Z 407.995,A -85,B 0,C 180,E1 -16320.641,E2 -16320.641} C_VEL
LIN {X 0,Y 302.024,Z 400.885,A -85,B 0,C 180,E1 -16323.49,E2 -16323.49} C_VEL
LIN {X 0,Y 300.026,Z 391.165,A -85,B 0,C 180,E1 -16327.52,E2 -16327.52} C_VEL
LIN {X 0,Y 298.433,Z 383.312,A -85,B 0,C 180,E1 -16330.985,E2 -16330.985} C_VEL
LIN {X 0,Y 298.426,Z 383.31,A -85,B 0,C 180,E1 -16333.109,E2 -16333.109} C_VEL
LIN {X 0,Y 298.403,Z 383.311,A -85,B 0,C 180,E1 -16336.921,E2 -16336.921} C_VEL
LIN {X 0,Y 298.416,Z 383.31,A -85,B 0,C 180,E1 -16341.003,E2 -16341.003} C_VEL
LIN {X 0,Y 298.433,Z 383.312,A -85,B 0,C 180,E1 -16343.932,E2 -16343.932} C_VEL
LIN {X 0,Y 298.395,Z 383.317,A -85,B 0,C 180,E1 -16347.983,E2 -16347.983} C_VEL
LIN {X 0,Y 298.459,Z 383.31,A -85,B 0,C 180,E1 -16351.904,E2 -16351.904} C_VEL
LIN {X 0,Y 298.486,Z 383.301,A -85,B 0,C 180,E1 -16354.924,E2 -16354.924} C_VEL
LIN {X 0,Y 298.451,Z 383.307,A -85,B 0,C 180,E1 -16359.315,E2 -16359.315} C_VEL
LIN {X 0,Y 298.538,Z 383.296,A -85,B 0,C 180,E1 -16362.179,E2 -16362.179} C_VEL
LIN {X 0,Y 298.594,Z 383.288,A -85,B 0,C 180,E1 -16364.995,E2 -16364.995} C_VEL
LIN {X 0,Y 298.594,Z 383.289,A -85,B 0,C 180,E1 -16369.147,E2 -16369.147} C_VEL
LIN {X 0,Y 298.759,Z 383.27,A -85,B 0,C 180,E1 -16371.886,E2 -16371.886} C_VEL
LIN {X 0,Y 298.662,Z 383.279,A -85,B 0,C 180,E1 -16374.599,E2 -16374.599} C_VEL
LIN {X 0,Y 298.927,Z 383.246,A -85,B 0,C 180,E1 -16378.653,E2 -16378.653} C_VEL
LIN {X 0,Y 298.924,Z 383.25,A -85,B 0,C 180,E1 -16381.347,E2 -16381.347} C_VEL
LIN {X 0,Y 298.799,Z 383.263,A -85,B 0,C 180,E1 -16386.754,E2 -16386.754} C_VEL
LIN {X 0,Y 298.682,Z 383.281,A -85,B 0,C 180,E1 -16389.48,E2 -16389.48} C_VEL
LIN {X 0,Y 298.555,Z 383.295,A -85,B 0,C 180,E1 -16393.615,E2 -16393.615} C_VEL
LIN {X 0,Y 298.55,Z 383.293,A -85,B 0,C 180,E1 -16396.409,E2 -16396.409} C_VEL
LIN {X 0,Y 298.512,Z 383.3,A -85,B 0,C 180,E1 -16399.655,E2 -16399.655} C_VEL
LIN {X 0,Y 298.458,Z 383.306,A -85,B 0,C 180,E1 -16403.598,E2 -16403.598} C_VEL
LIN {X 0,Y 298.49,Z 383.302,A -85,B 0,C 180,E1 -16406.574,E2 -16406.574} C_VEL
LIN {X 0,Y 298.422,Z 383.31,A -85,B 0,C 180,E1 -16409.641,E2 -16409.641} C_VEL
LIN {X 0,Y 298.396,Z 383.316,A -85,B 0,C 180,E1 -16412.8,E2 -16412.8} C_VEL
LIN {X 0,Y 298.447,Z 383.311,A -85,B 0,C 180,E1 -16416.808,E2 -16416.808} C_VEL
LIN {X 0,Y 298.388,Z 383.316,A -85,B 0,C 180,E1 -16421.088,E2 -16421.088} C_VEL
LIN {X 0,Y 298.389,Z 383.316,A -85,B 0,C 180,E1 -16425.042,E2 -16425.042} C_VEL
LIN {X 0,Y 298.389,Z 383.316,A -85,B 0,C 180,E1 -16428.912,E2 -16428.912} C_VEL
LIN {X 0,Y 298.466,Z 383.305,A -85,B 0,C 180,E1 -16433.188,E2 -16433.188} C_VEL
LIN {X 0,Y 298.396,Z 383.313,A -85,B 0,C 180,E1 -16437.2,E2 -16437.2} C_VEL
LIN {X 0,Y 298.428,Z 383.312,A -85,B 0,C 180,E1 -16440.617,E2 -16440.617} C_VEL
LIN {X 0,Y 298.48,Z 383.302,A -85,B 0,C 180,E1 -16443.477,E2 -16443.477} C_VEL
LIN {X 0,Y 298.437,Z 383.31,A -85,B 0,C 180,E1 -16446.697,E2 -16446.697} C_VEL
LIN {X 0,Y 298.545,Z 383.296,A -85,B 0,C 180,E1 -16450.757,E2 -16450.757} C_VEL
LIN {X 0,Y 298.615,Z 383.285,A -85,B 0,C 180,E1 -16454.996,E2 -16454.996} C_VEL
LIN {X 0,Y 298.596,Z 383.287,A -85,B 0,C 180,E1 -16459.147,E2 -16459.147} C_VEL
LIN {X 0,Y 298.757,Z 383.271,A -85,B 0,C 180,E1 -16461.886,E2 -16461.886} C_VEL
LIN {X 0,Y 298.66,Z 383.28,A -85,B 0,C 180,E1 -16464.599,E2 -16464.599} C_VEL
LIN {X 0,Y 298.926,Z 383.247,A -85,B 0,C 180,E1 -16468.653,E2 -16468.653} C_VEL
LIN {X 0,Y 298.926,Z 383.247,A -85,B 0,C 180,E1 -16471.347,E2 -16471.347} C_VEL
LIN {X 0,Y 298.79,Z 383.264,A -85,B 0,C 180,E1 -16476.754,E2 -16476.754} C_VEL
LIN {X 0,Y 298.638,Z 383.285,A -85,B 0,C 180,E1 -16479.482,E2 -16479.482} C_VEL
LIN {X 0,Y 298.555,Z 383.296,A -85,B 0,C 180,E1 -16483.616,E2 -16483.616} C_VEL
LIN {X 0,Y 298.552,Z 383.294,A -85,B 0,C 180,E1 -16486.409,E2 -16486.409} C_VEL
LIN {X 0,Y 298.514,Z 383.303,A -85,B 0,C 180,E1 -16489.655,E2 -16489.655} C_VEL
LIN {X 0,Y 298.46,Z 383.31,A -85,B 0,C 180,E1 -16493.598,E2 -16493.598} C_VEL
LIN {X 0,Y 298.489,Z 383.301,A -85,B 0,C 180,E1 -16496.575,E2 -16496.575} C_VEL
LIN {X 0,Y 298.419,Z 383.313,A -85,B 0,C 180,E1 -16499.642,E2 -16499.642} C_VEL
LIN {X 0,Y 298.397,Z 383.313,A -85,B 0,C 180,E1 -16502.8,E2 -16502.8} C_VEL
LIN {X 0,Y 298.467,Z 383.305,A -85,B 0,C 180,E1 -16506.813,E2 -16506.813} C_VEL
LIN {X 0,Y 298.391,Z 383.316,A -85,B 0,C 180,E1 -16511.088,E2 -16511.088} C_VEL
LIN {X 0,Y 298.391,Z 383.317,A -85,B 0,C 180,E1 -16515.042,E2 -16515.042} C_VEL
LIN {X 0,Y 298.39,Z 383.316,A -85,B 0,C 180,E1 -16518.912,E2 -16518.912} C_VEL
LIN {X 0,Y 298.45,Z 383.31,A -85,B 0,C 180,E1 -16523.192,E2 -16523.192} C_VEL
LIN {X 0,Y 298.588,Z 383.293,A -85,B 0,C 180,E1 -16527.925,E2 -16527.925} C_VEL
LIN {X 0,Y 298.8,Z 384.356,A -85,B 0,C 180,E1 -16528.838,E2 -16528.838} C_VEL
LIN {X 0,Y 298.606,Z 388.96,A -85,B 0,C 180,E1 -16531.919,E2 -16531.919} C_VEL
LIN {X 0,Y 298.161,Z 394.652,A -85,B 0,C 180,E1 -16535.638,E2 -16535.638} C_VEL
LIN {X 0,Y 297.792,Z 401.404,A -85,B 0,C 180,E1 -16539.989,E2 -16539.989} C_VEL
LIN {X 0,Y 297.461,Z 408.195,A -85,B 0,C 180,E1 -16544.234,E2 -16544.234} C_VEL
LIN {X 0,Y 297.275,Z 413.379,A -85,B 0,C 180,E1 -16547.412,E2 -16547.412} C_VEL
LIN {X 0,Y 298.475,Z 425.598,A -85,B 0,C 180,E1 -16548.368,E2 -16548.368} C_VEL
LIN {X 0,Y 299.173,Z 432.092,A -85,B 0,C 180,E1 -16548.997,E2 -16548.997} C_VEL
LIN {X 0,Y 298.677,Z 442.24,A -85,B 0,C 180,E1 -16550.177,E2 -16550.177} C_VEL
LIN {X 0,Y 298.281,Z 451.438,A -85,B 0,C 180,E1 -16551.532,E2 -16551.532} C_VEL
LIN {X 0,Y 297.979,Z 459.22,A -85,B 0,C 180,E1 -16552.961,E2 -16552.961} C_VEL
LIN {X 0,Y 297.694,Z 466.269,A -85,B 0,C 180,E1 -16554.581,E2 -16554.581} C_VEL
LIN {X 0,Y 297.332,Z 472.083,A -85,B 0,C 180,E1 -16556.273,E2 -16556.273} C_VEL
LIN {X 0,Y 297.225,Z 476.586,A -85,B 0,C 180,E1 -16557.967,E2 -16557.967} C_VEL
LIN {X 0,Y 297.278,Z 480.5,A -85,B 0,C 180,E1 -16560,E2 -16560} C_VEL
LIN {X 0,Y 297.39,Z 481.851,A -85,B 0,C 180,E1 -16561.035,E2 -16561.035} C_VEL
LIN {X 0,Y 296.944,Z 483.153,A -85,B 0,C 180,E1 -16562.146,E2 -16562.146} C_VEL
LIN {X 0,Y 294.651,Z 484.532,A -85,B 0,C 180,E1 -16564.001,E2 -16564.001} C_VEL
LIN {X 0,Y 292.911,Z 484.754,A -85,B 0,C 180,E1 -16565.512,E2 -16565.512} C_VEL
LIN {X 0,Y 292.517,Z 484.298,A -85,B 0,C 180,E1 -16566.661,E2 -16566.661} C_VEL
LIN {X 0,Y 292.675,Z 484.009,A -85,B 0,C 180,E1 -16567.041,E2 -16567.041} C_VEL
LIN {X 0,Y 293.54,Z 482.957,A -85,B 0,C 180,E1 -16568.259,E2 -16568.259} C_VEL
LIN {X 0,Y 295.312,Z 480.003,A -85,B 0,C 180,E1 -16570.282,E2 -16570.282} C_VEL
LIN {X 0,Y 297.29,Z 475.607,A -85,B 0,C 180,E1 -16572.284,E2 -16572.284} C_VEL
LIN {X 0,Y 299.652,Z 469.602,A -85,B 0,C 180,E1 -16574.257,E2 -16574.257} C_VEL
LIN {X 0,Y 301.891,Z 463.096,A -85,B 0,C 180,E1 -16575.875,E2 -16575.875} C_VEL
LIN {X 0,Y 303.798,Z 456.982,A -85,B 0,C 180,E1 -16577.106,E2 -16577.106} C_VEL
LIN {X 0,Y 303.925,Z 452.599,A -85,B 0,C 180,E1 -16578.074,E2 -16578.074} C_VEL
LIN {X 0,Y 302.982,Z 445.061,A -85,B 0,C 180,E1 -16579.736,E2 -16579.736} C_VEL
LIN {X 0,Y 301.117,Z 437.037,A -85,B 0,C 180,E1 -16581.508,E2 -16581.508} C_VEL
LIN {X 0,Y 298.446,Z 429.214,A -85,B 0,C 180,E1 -16583.306,E2 -16583.306} C_VEL
LIN {X 0,Y 295.697,Z 422.138,A -85,B 0,C 180,E1 -16584.953,E2 -16584.953} C_VEL
LIN {X 0,Y 297.038,Z 418.951,A -85,B 0,C 180,E1 -16588.903,E2 -16588.903} C_VEL
LIN {X 0,Y 297.931,Z 417.078,A -85,B 0,C 180,E1 -16591.873,E2 -16591.873} C_VEL
LIN {X 0,Y 298.359,Z 416,A -85,B 0,C 180,E1 -16594.467,E2 -16594.467} C_VEL
LIN {X 0,Y 298.661,Z 415.326,A -85,B 0,C 180,E1 -16597.722,E2 -16597.722} C_VEL
LIN {X 0,Y 299.006,Z 415.426,A -85,B 0,C 180,E1 -16601.223,E2 -16601.223} C_VEL
LIN {X 0,Y 299.261,Z 415.911,A -85,B 0,C 180,E1 -16603.279,E2 -16603.279} C_VEL
LIN {X 0,Y 299.822,Z 417.763,A -85,B 0,C 180,E1 -16607.173,E2 -16607.173} C_VEL
LIN {X 0,Y 300.37,Z 420.408,A -85,B 0,C 180,E1 -16610.546,E2 -16610.546} C_VEL
LIN {X 0,Y 301.3,Z 424.463,A -85,B 0,C 180,E1 -16614.328,E2 -16614.328} C_VEL
LIN {X 0,Y 301.786,Z 426.692,A -85,B 0,C 180,E1 -16616.019,E2 -16616.019} C_VEL
LIN {X 0,Y 301.663,Z 429.216,A -85,B 0,C 180,E1 -16617.598,E2 -16617.598} C_VEL
LIN {X 0,Y 299.927,Z 433.505,A -85,B 0,C 180,E1 -16619.749,E2 -16619.749} C_VEL
LIN {X 0,Y 299.302,Z 435.429,A -85,B 0,C 180,E1 -16620.557,E2 -16620.557} C_VEL
LIN {X 0,Y 302.018,Z 447.429,A -85,B 0,C 180,E1 -16622.162,E2 -16622.162} C_VEL
LIN {X 0,Y 303.49,Z 457.75,A -85,B 0,C 180,E1 -16623.526,E2 -16623.526} C_VEL
LIN {X 0,Y 304.011,Z 467.546,A -85,B 0,C 180,E1 -16624.819,E2 -16624.819} C_VEL
LIN {X 0,Y 303.428,Z 477.008,A -85,B 0,C 180,E1 -16626.088,E2 -16626.088} C_VEL
LIN {X 0,Y 301.529,Z 487.263,A -85,B 0,C 180,E1 -16627.563,E2 -16627.563} C_VEL
LIN {X 0,Y 298.585,Z 497.779,A -85,B 0,C 180,E1 -16629.325,E2 -16629.325} C_VEL
LIN {X 0,Y 295.982,Z 507.065,A -85,B 0,C 180,E1 -16631.303,E2 -16631.303} C_VEL
LIN {X 0,Y 293.821,Z 514.642,A -85,B 0,C 180,E1 -16633.319,E2 -16633.319} C_VEL
LIN {X 0,Y 292.264,Z 520.798,A -85,B 0,C 180,E1 -16635.375,E2 -16635.375} C_VEL
LIN {X 0,Y 290.962,Z 525.784,A -85,B 0,C 180,E1 -16637.444,E2 -16637.444} C_VEL
LIN {X 0,Y 290.189,Z 529.693,A -85,B 0,C 180,E1 -16639.534,E2 -16639.534} C_VEL
LIN {X 0,Y 289.869,Z 532.616,A -85,B 0,C 180,E1 -16641.635,E2 -16641.635} C_VEL
LIN {X 0,Y 289.848,Z 534.64,A -85,B 0,C 180,E1 -16643.793,E2 -16643.793} C_VEL
LIN {X 0,Y 289.894,Z 535.628,A -85,B 0,C 180,E1 -16645.829,E2 -16645.829} C_VEL
LIN {X 0,Y 290.134,Z 535.823,A -85,B 0,C 180,E1 -16647.223,E2 -16647.223} C_VEL
LIN {X 0,Y 290.362,Z 535.547,A -85,B 0,C 180,E1 -16648.613,E2 -16648.613} C_VEL
LIN {X 0,Y 290.382,Z 534.808,A -85,B 0,C 180,E1 -16650,E2 -16650} C_VEL
LIN {X 0,Y 290.448,Z 533.644,A -85,B 0,C 180,E1 -16651.386,E2 -16651.386} C_VEL
LIN {X 0,Y 290.431,Z 530.932,A -85,B 0,C 180,E1 -16653.468,E2 -16653.468} C_VEL
LIN {X 0,Y 290.368,Z 526.999,A -85,B 0,C 180,E1 -16655.556,E2 -16655.556} C_VEL
LIN {X 0,Y 290.377,Z 521.749,A -85,B 0,C 180,E1 -16657.649,E2 -16657.649} C_VEL
LIN {X 0,Y 290.475,Z 514.981,A -85,B 0,C 180,E1 -16659.751,E2 -16659.751} C_VEL
LIN {X 0,Y 290.91,Z 506.332,A -85,B 0,C 180,E1 -16661.85,E2 -16661.85} C_VEL
LIN {X 0,Y 291.477,Z 497.341,A -85,B 0,C 180,E1 -16663.597,E2 -16663.597} C_VEL
LIN {X 0,Y 292.328,Z 486.053,A -85,B 0,C 180,E1 -16665.334,E2 -16665.334} C_VEL
LIN {X 0,Y 293.088,Z 475.469,A -85,B 0,C 180,E1 -16666.614,E2 -16666.614} C_VEL
LIN {X 0,Y 292.699,Z 465.726,A -85,B 0,C 180,E1 -16667.556,E2 -16667.556} C_VEL
LIN {X 0,Y 291.835,Z 452.924,A -85,B 0,C 180,E1 -16668.517,E2 -16668.517} C_VEL
LIN {X 0,Y 291.414,Z 438.916,A -85,B 0,C 180,E1 -16669.275,E2 -16669.275} C_VEL
LIN {X 0,Y 293.247,Z 425.394,A -85,B 0,C 180,E1 -16674.396,E2 -16674.396} C_VEL
LIN {X 0,Y 295.524,Z 412.833,A -85,B 0,C 180,E1 -16679.177,E2 -16679.177} C_VEL
LIN {X 0,Y 296.256,Z 409.139,A -85,B 0,C 180,E1 -16680.585,E2 -16680.585} C_VEL
LIN {X 0,Y 295.612,Z 404.767,A -85,B 0,C 180,E1 -16682.339,E2 -16682.339} C_VEL
LIN {X 0,Y 293.427,Z 394.276,A -85,B 0,C 180,E1 -16686.783,E2 -16686.783} C_VEL
LIN {X 0,Y 291.68,Z 385.687,A -85,B 0,C 180,E1 -16690.584,E2 -16690.584} C_VEL
LIN {X 0,Y 291.38,Z 384.191,A -85,B 0,C 180,E1 -16691.338,E2 -16691.338} C_VEL
LIN {X 0,Y 291.314,Z 384.195,A -85,B 0,C 180,E1 -16695.603,E2 -16695.603} C_VEL
LIN {X 0,Y 291.336,Z 384.192,A -85,B 0,C 180,E1 -16699.358,E2 -16699.358} C_VEL
LIN {X 0,Y 291.425,Z 384.181,A -85,B 0,C 180,E1 -16702.922,E2 -16702.922} C_VEL
LIN {X 0,Y 291.345,Z 384.194,A -85,B 0,C 180,E1 -16706.302,E2 -16706.302} C_VEL
LIN {X 0,Y 291.384,Z 384.189,A -85,B 0,C 180,E1 -16710.261,E2 -16710.261} C_VEL
LIN {X 0,Y 291.417,Z 384.184,A -85,B 0,C 180,E1 -16714.272,E2 -16714.272} C_VEL
LIN {X 0,Y 291.382,Z 384.187,A -85,B 0,C 180,E1 -16717.3,E2 -16717.3} C_VEL
LIN {X 0,Y 291.459,Z 384.178,A -85,B 0,C 180,E1 -16720.27,E2 -16720.27} C_VEL
LIN {X 0,Y 291.555,Z 384.165,A -85,B 0,C 180,E1 -16724.624,E2 -16724.624} C_VEL
LIN {X 0,Y 291.538,Z 384.167,A -85,B 0,C 180,E1 -16728.881,E2 -16728.881} C_VEL
LIN {X 0,Y 291.71,Z 384.15,A -85,B 0,C 180,E1 -16731.689,E2 -16731.689} C_VEL
LIN {X 0,Y 291.632,Z 384.155,A -85,B 0,C 180,E1 -16734.468,E2 -16734.468} C_VEL
LIN {X 0,Y 291.893,Z 384.122,A -85,B 0,C 180,E1 -16738.62,E2 -16738.62} C_VEL
LIN {X 0,Y 291.891,Z 384.127,A -85,B 0,C 180,E1 -16741.38,E2 -16741.38} C_VEL
LIN {X 0,Y 291.747,Z 384.142,A -85,B 0,C 180,E1 -16746.918,E2 -16746.918} C_VEL
LIN {X 0,Y 291.63,Z 384.157,A -85,B 0,C 180,E1 -16749.712,E2 -16749.712} C_VEL
LIN {X 0,Y 291.524,Z 384.169,A -85,B 0,C 180,E1 -16753.95,E2 -16753.95} C_VEL
LIN {X 0,Y 291.488,Z 384.174,A -85,B 0,C 180,E1 -16756.818,E2 -16756.818} C_VEL
LIN {X 0,Y 291.451,Z 384.178,A -85,B 0,C 180,E1 -16759.875,E2 -16759.875} C_VEL
LIN {X 0,Y 291.401,Z 384.184,A -85,B 0,C 180,E1 -16764.205,E2 -16764.205} C_VEL
LIN {X 0,Y 291.423,Z 384.184,A -85,B 0,C 180,E1 -16767.272,E2 -16767.272} C_VEL
LIN {X 0,Y 291.338,Z 384.193,A -85,B 0,C 180,E1 -16770.437,E2 -16770.437} C_VEL
